LIN {X 0,Y 369.158,Z 304.498,A -85,B 0,C 180,E1 -12863.442,E2 -12863.442} C_VEL
LIN {X 0,Y 369.295,Z 304.483,A -85,B 0,C 180,E1 -12867.819,E2 -12867.819} C_VEL
LIN {X 0,Y 369.206,Z 304.491,A -85,B 0,C 180,E1 -12871.091,E2 -12871.091} C_VEL
LIN {X 0,Y 369.294,Z 304.487,A -85,B 0,C 180,E1 -12872.182,E2 -12872.182} C_VEL
LIN {X 0,Y 369.16,Z 304.501,A -85,B 0,C 180,E1 -12876.56,E2 -12876.56} C_VEL
LIN {X 0,Y 369.039,Z 304.513,A -85,B 0,C 180,E1 -12879.87,E2 -12879.87} C_VEL
LIN {X 0,Y 369.006,Z 304.516,A -85,B 0,C 180,E1 -12883.749,E2 -12883.749} C_VEL
LIN {X 0,Y 368.958,Z 304.522,A -85,B 0,C 180,E1 -12887.745,E2 -12887.745} C_VEL
LIN {X 0,Y 368.914,Z 304.532,A -85,B 0,C 180,E1 -12891.221,E2 -12891.221} C_VEL
LIN {X 0,Y 368.962,Z 304.615,A -85,B 0,C 180,E1 -12893.171,E2 -12893.171} C_VEL
LIN {X 0,Y 370.807,Z 314.362,A -85,B 0,C 180,E1 -12895.845,E2 -12895.845} C_VEL
LIN {X 0,Y 373.154,Z 322.489,A -85,B 0,C 180,E1 -12896.158,E2 -12896.158} C_VEL
LIN {X 0,Y 376.257,Z 338.846,A -85,B 0,C 180,E1 -12896.672,E2 -12896.672} C_VEL
LIN {X 0,Y 374.9,Z 409.964,A -85,B 0,C 180,E1 -12898.135,E2 -12898.135} C_VEL
LIN {X 0,Y 374.138,Z 415.804,A -85,B 0,C 180,E1 -12898.226,E2 -12898.226} C_VEL
LIN {X 0,Y 371.004,Z 425.22,A -85,B 0,C 180,E1 -12898.352,E2 -12898.352} C_VEL
LIN {X 0,Y 367.894,Z 434.497,A -85,B 0,C 180,E1 -12898.587,E2 -12898.587} C_VEL
LIN {X 0,Y 367.116,Z 440.104,A -85,B 0,C 180,E1 -12898.842,E2 -12898.842} C_VEL
LIN {X 0,Y 366.35,Z 452.424,A -85,B 0,C 180,E1 -12899.603,E2 -12899.603} C_VEL
LIN {X 0,Y 365.516,Z 464,A -85,B 0,C 180,E1 -12900.548,E2 -12900.548} C_VEL
LIN {X 0,Y 364.656,Z 474.566,A -85,B 0,C 180,E1 -12901.646,E2 -12901.646} C_VEL
LIN {X 0,Y 363.853,Z 484.377,A -85,B 0,C 180,E1 -12902.905,E2 -12902.905} C_VEL
LIN {X 0,Y 362.988,Z 493.439,A -85,B 0,C 180,E1 -12904.327,E2 -12904.327} C_VEL
LIN {X 0,Y 362.136,Z 501.792,A -85,B 0,C 180,E1 -12905.949,E2 -12905.949} C_VEL
LIN {X 0,Y 361.431,Z 509.337,A -85,B 0,C 180,E1 -12907.799,E2 -12907.799} C_VEL
LIN {X 0,Y 361.041,Z 514.472,A -85,B 0,C 180,E1 -12909.389,E2 -12909.389} C_VEL
LIN {X 0,Y 360.728,Z 518.553,A -85,B 0,C 180,E1 -12910.99,E2 -12910.99} C_VEL
LIN {X 0,Y 360.364,Z 522.397,A -85,B 0,C 180,E1 -12913.047,E2 -12913.047} C_VEL
LIN {X 0,Y 360.207,Z 524.3,A -85,B 0,C 180,E1 -12914.62,E2 -12914.62} C_VEL
LIN {X 0,Y 360.172,Z 525.614,A -85,B 0,C 180,E1 -12916.925,E2 -12916.925} C_VEL
LIN {X 0,Y 360.174,Z 525.57,A -85,B 0,C 180,E1 -12918.437,E2 -12918.437} C_VEL
LIN {X 0,Y 360.258,Z 524.77,A -85,B 0,C 180,E1 -12919.926,E2 -12919.926} C_VEL
LIN {X 0,Y 360.63,Z 522.252,A -85,B 0,C 180,E1 -12922.129,E2 -12922.129} C_VEL
LIN {X 0,Y 361.086,Z 518.191,A -85,B 0,C 180,E1 -12924.274,E2 -12924.274} C_VEL
LIN {X 0,Y 361.701,Z 513.027,A -85,B 0,C 180,E1 -12926.201,E2 -12926.201} C_VEL
LIN {X 0,Y 362.518,Z 506.261,A -85,B 0,C 180,E1 -12928.11,E2 -12928.11} C_VEL
LIN {X 0,Y 363.46,Z 498.606,A -85,B 0,C 180,E1 -12929.818,E2 -12929.818} C_VEL
LIN {X 0,Y 364.603,Z 489.19,A -85,B 0,C 180,E1 -12931.477,E2 -12931.477} C_VEL
LIN {X 0,Y 365.673,Z 479.6,A -85,B 0,C 180,E1 -12932.841,E2 -12932.841} C_VEL
LIN {X 0,Y 366.845,Z 468.816,A -85,B 0,C 180,E1 -12934.07,E2 -12934.07} C_VEL
LIN {X 0,Y 367.921,Z 456.729,A -85,B 0,C 180,E1 -12935.15,E2 -12935.15} C_VEL
LIN {X 0,Y 368.805,Z 445.404,A -85,B 0,C 180,E1 -12935.928,E2 -12935.928} C_VEL
LIN {X 0,Y 369.489,Z 432.429,A -85,B 0,C 180,E1 -12936.586,E2 -12936.586} C_VEL
LIN {X 0,Y 369.985,Z 418.805,A -85,B 0,C 180,E1 -12937.027,E2 -12937.027} C_VEL
LIN {X 0,Y 371.953,Z 339.841,A -85,B 0,C 180,E1 -12938.741,E2 -12938.741} C_VEL
LIN {X 0,Y 369.024,Z 326.317,A -85,B 0,C 180,E1 -12939.288,E2 -12939.288} C_VEL
LIN {X 0,Y 364.19,Z 314.682,A -85,B 0,C 180,E1 -12939.968,E2 -12939.968} C_VEL
LIN {X 0,Y 361.958,Z 305.404,A -85,B 0,C 180,E1 -12942.326,E2 -12942.326} C_VEL
LIN {X 0,Y 362.001,Z 305.397,A -85,B 0,C 180,E1 -12946.101,E2 -12946.101} C_VEL
LIN {X 0,Y 362.033,Z 305.389,A -85,B 0,C 180,E1 -12949.938,E2 -12949.938} C_VEL
LIN {X 0,Y 362.153,Z 305.376,A -85,B 0,C 180,E1 -12952.192,E2 -12952.192} C_VEL
LIN {X 0,Y 362.118,Z 305.379,A -85,B 0,C 180,E1 -12954.431,E2 -12954.431} C_VEL
LIN {X 0,Y 362.282,Z 305.358,A -85,B 0,C 180,E1 -12957.776,E2 -12957.776} C_VEL
LIN {X 0,Y 362.428,Z 305.34,A -85,B 0,C 180,E1 -12960,E2 -12960} C_VEL
LIN {X 0,Y 362.282,Z 305.36,A -85,B 0,C 180,E1 -12962.223,E2 -12962.223} C_VEL
LIN {X 0,Y 362.141,Z 305.368,A -85,B 0,C 180,E1 -12966.687,E2 -12966.687} C_VEL
LIN {X 0,Y 362.033,Z 305.384,A -85,B 0,C 180,E1 -12970.062,E2 -12970.062} C_VEL
LIN {X 0,Y 362,Z 305.386,A -85,B 0,C 180,E1 -12973.898,E2 -12973.898} C_VEL
LIN {X 0,Y 361.93,Z 305.394,A -85,B 0,C 180,E1 -12976.934,E2 -12976.934} C_VEL
LIN {X 0,Y 361.888,Z 305.402,A -85,B 0,C 180,E1 -12980.461,E2 -12980.461} C_VEL
LIN {X 0,Y 361.895,Z 305.401,A -85,B 0,C 180,E1 -12984.113,E2 -12984.113} C_VEL
LIN {X 0,Y 361.943,Z 305.399,A -85,B 0,C 180,E1 -12986.721,E2 -12986.721} C_VEL
LIN {X 0,Y 361.875,Z 305.407,A -85,B 0,C 180,E1 -12990.328,E2 -12990.328} C_VEL
LIN {X 0,Y 361.856,Z 305.408,A -85,B 0,C 180,E1 -12994.28,E2 -12994.28} C_VEL
LIN {X 0,Y 361.865,Z 305.407,A -85,B 0,C 180,E1 -12997.223,E2 -12997.223} C_VEL
LIN {X 0,Y 361.837,Z 305.41,A -85,B 0,C 180,E1 -13000.755,E2 -13000.755} C_VEL
LIN {X 0,Y 361.819,Z 305.415,A -85,B 0,C 180,E1 -13004.368,E2 -13004.368} C_VEL
LIN {X 0,Y 361.838,Z 305.413,A -85,B 0,C 180,E1 -13007.568,E2 -13007.568} C_VEL
LIN {X 0,Y 361.87,Z 305.41,A -85,B 0,C 180,E1 -13010.973,E2 -13010.973} C_VEL
LIN {X 0,Y 361.876,Z 305.413,A -85,B 0,C 180,E1 -13014.655,E2 -13014.655} C_VEL
LIN {X 0,Y 361.84,Z 305.417,A -85,B 0,C 180,E1 -13018.37,E2 -13018.37} C_VEL
LIN {X 0,Y 361.934,Z 305.557,A -85,B 0,C 180,E1 -13019.41,E2 -13019.41} C_VEL
LIN {X 0,Y 364.728,Z 317.304,A -85,B 0,C 180,E1 -13022.422,E2 -13022.422} C_VEL
LIN {X 0,Y 366.195,Z 325.557,A -85,B 0,C 180,E1 -13024.425,E2 -13024.425} C_VEL
LIN {X 0,Y 365.204,Z 338.309,A -85,B 0,C 180,E1 -13027.185,E2 -13027.185} C_VEL
LIN {X 0,Y 369.361,Z 360.306,A -85,B 0,C 180,E1 -13028.032,E2 -13028.032} C_VEL
LIN {X 0,Y 371.307,Z 374.136,A -85,B 0,C 180,E1 -13028.503,E2 -13028.503} C_VEL
LIN {X 0,Y 369.57,Z 448.21,A -85,B 0,C 180,E1 -13030.127,E2 -13030.127} C_VEL
LIN {X 0,Y 368.75,Z 462.309,A -85,B 0,C 180,E1 -13030.661,E2 -13030.661} C_VEL
LIN {X 0,Y 367.815,Z 474.39,A -85,B 0,C 180,E1 -13031.334,E2 -13031.334} C_VEL
LIN {X 0,Y 366.667,Z 486.939,A -85,B 0,C 180,E1 -13032.285,E2 -13032.285} C_VEL
LIN {X 0,Y 365.455,Z 498.198,A -85,B 0,C 180,E1 -13033.377,E2 -13033.377} C_VEL
LIN {X 0,Y 364.303,Z 508.998,A -85,B 0,C 180,E1 -13034.706,E2 -13034.706} C_VEL
LIN {X 0,Y 363.353,Z 517.608,A -85,B 0,C 180,E1 -13036.008,E2 -13036.008} C_VEL
LIN {X 0,Y 362.265,Z 526.631,A -85,B 0,C 180,E1 -13037.678,E2 -13037.678} C_VEL
LIN {X 0,Y 361.447,Z 533.915,A -85,B 0,C 180,E1 -13039.355,E2 -13039.355} C_VEL
LIN {X 0,Y 360.915,Z 539.734,A -85,B 0,C 180,E1 -13041.037,E2 -13041.037} C_VEL
LIN {X 0,Y 360.591,Z 544.332,A -85,B 0,C 180,E1 -13042.721,E2 -13042.721} C_VEL
LIN {X 0,Y 360.383,Z 547.831,A -85,B 0,C 180,E1 -13044.404,E2 -13044.404} C_VEL
LIN {X 0,Y 360.365,Z 549.58,A -85,B 0,C 180,E1 -13045.525,E2 -13045.525} C_VEL
LIN {X 0,Y 360.302,Z 550.917,A -85,B 0,C 180,E1 -13046.645,E2 -13046.645} C_VEL
LIN {X 0,Y 360.297,Z 551.851,A -85,B 0,C 180,E1 -13047.764,E2 -13047.764} C_VEL
LIN {X 0,Y 360.369,Z 552.338,A -85,B 0,C 180,E1 -13048.882,E2 -13048.882} C_VEL
LIN {X 0,Y 360.424,Z 552.415,A -85,B 0,C 180,E1 -13049.999,E2 -13049.999} C_VEL
LIN {X 0,Y 360.385,Z 552.091,A -85,B 0,C 180,E1 -13051.117,E2 -13051.117} C_VEL
LIN {X 0,Y 360.304,Z 551.362,A -85,B 0,C 180,E1 -13052.235,E2 -13052.235} C_VEL
LIN {X 0,Y 360.305,Z 550.176,A -85,B 0,C 180,E1 -13053.354,E2 -13053.354} C_VEL
LIN {X 0,Y 360.364,Z 547.607,A -85,B 0,C 180,E1 -13055.034,E2 -13055.034} C_VEL
LIN {X 0,Y 360.496,Z 543.988,A -85,B 0,C 180,E1 -13056.717,E2 -13056.717} C_VEL
LIN {X 0,Y 360.747,Z 539.221,A -85,B 0,C 180,E1 -13058.401,E2 -13058.401} C_VEL
LIN {X 0,Y 361.25,Z 532.028,A -85,B 0,C 180,E1 -13060.366,E2 -13060.366} C_VEL
LIN {X 0,Y 361.951,Z 524.189,A -85,B 0,C 180,E1 -13062.047,E2 -13062.047} C_VEL
LIN {X 0,Y 362.661,Z 516.147,A -85,B 0,C 180,E1 -13063.446,E2 -13063.446} C_VEL
LIN {X 0,Y 363.64,Z 505.802,A -85,B 0,C 180,E1 -13064.908,E2 -13064.908} C_VEL
LIN {X 0,Y 364.478,Z 495.426,A -85,B 0,C 180,E1 -13066.091,E2 -13066.091} C_VEL
LIN {X 0,Y 365.404,Z 484.808,A -85,B 0,C 180,E1 -13067.055,E2 -13067.055} C_VEL
LIN {X 0,Y 366.352,Z 472.083,A -85,B 0,C 180,E1 -13067.946,E2 -13067.946} C_VEL
LIN {X 0,Y 367.178,Z 459.469,A -85,B 0,C 180,E1 -13068.59,E2 -13068.59} C_VEL
LIN {X 0,Y 367.723,Z 446.201,A -85,B 0,C 180,E1 -13069.032,E2 -13069.032} C_VEL
LIN {X 0,Y 368.945,Z 372.876,A -85,B 0,C 180,E1 -13070.593,E2 -13070.593} C_VEL
LIN {X 0,Y 364.224,Z 340.195,A -85,B 0,C 180,E1 -13071.604,E2 -13071.604} C_VEL
LIN {X 0,Y 365.627,Z 325.106,A -85,B 0,C 180,E1 -13075.016,E2 -13075.016} C_VEL
LIN {X 0,Y 364.637,Z 318.571,A -85,B 0,C 180,E1 -13076.601,E2 -13076.601} C_VEL
LIN {X 0,Y 362.081,Z 306.333,A -85,B 0,C 180,E1 -13079.706,E2 -13079.706} C_VEL
LIN {X 0,Y 361.886,Z 305.409,A -85,B 0,C 180,E1 -13079.949,E2 -13079.949} C_VEL
LIN {X 0,Y 361.858,Z 305.409,A -85,B 0,C 180,E1 -13083.369,E2 -13083.369} C_VEL
LIN {X 0,Y 361.864,Z 305.406,A -85,B 0,C 180,E1 -13087.017,E2 -13087.017} C_VEL
LIN {X 0,Y 361.851,Z 305.409,A -85,B 0,C 180,E1 -13089.861,E2 -13089.861} C_VEL
LIN {X 0,Y 361.832,Z 305.412,A -85,B 0,C 180,E1 -13092.828,E2 -13092.828} C_VEL
LIN {X 0,Y 361.816,Z 305.413,A -85,B 0,C 180,E1 -13095.946,E2 -13095.946} C_VEL
LIN {X 0,Y 361.833,Z 305.41,A -85,B 0,C 180,E1 -13099.244,E2 -13099.244} C_VEL
LIN {X 0,Y 361.867,Z 305.411,A -85,B 0,C 180,E1 -13102.775,E2 -13102.775} C_VEL
LIN {X 0,Y 361.849,Z 305.407,A -85,B 0,C 180,E1 -13105.719,E2 -13105.719} C_VEL
LIN {X 0,Y 361.868,Z 305.405,A -85,B 0,C 180,E1 -13109.672,E2 -13109.672} C_VEL
LIN {X 0,Y 361.948,Z 305.397,A -85,B 0,C 180,E1 -13113.475,E2 -13113.475} C_VEL
LIN {X 0,Y 361.885,Z 305.41,A -85,B 0,C 180,E1 -13117.144,E2 -13117.144} C_VEL
LIN {X 0,Y 361.915,Z 305.401,A -85,B 0,C 180,E1 -13120.724,E2 -13120.724} C_VEL
LIN {X 0,Y 361.94,Z 305.396,A -85,B 0,C 180,E1 -13124.226,E2 -13124.226} C_VEL
LIN {X 0,Y 361.993,Z 305.39,A -85,B 0,C 180,E1 -13126.528,E2 -13126.528} C_VEL
LIN {X 0,Y 362.025,Z 305.387,A -85,B 0,C 180,E1 -13129.938,E2 -13129.938} C_VEL
LIN {X 0,Y 362.145,Z 305.371,A -85,B 0,C 180,E1 -13132.193,E2 -13132.193} C_VEL
LIN {X 0,Y 362.112,Z 305.375,A -85,B 0,C 180,E1 -13134.431,E2 -13134.431} C_VEL
LIN {X 0,Y 362.274,Z 305.36,A -85,B 0,C 180,E1 -13137.777,E2 -13137.777} C_VEL
LIN {X 0,Y 362.42,Z 305.34,A -85,B 0,C 180,E1 -13140,E2 -13140} C_VEL
LIN {X 0,Y 362.275,Z 305.357,A -85,B 0,C 180,E1 -13142.224,E2 -13142.224} C_VEL
LIN {X 0,Y 362.134,Z 305.372,A -85,B 0,C 180,E1 -13146.687,E2 -13146.687} C_VEL
LIN {X 0,Y 362.026,Z 305.392,A -85,B 0,C 180,E1 -13150.063,E2 -13150.063} C_VEL
LIN {X 0,Y 361.993,Z 305.394,A -85,B 0,C 180,E1 -13153.899,E2 -13153.899} C_VEL
LIN {X 0,Y 361.963,Z 305.397,A -85,B 0,C 180,E1 -13157.939,E2 -13157.939} C_VEL
LIN {X 0,Y 361.856,Z 305.407,A -85,B 0,C 180,E1 -13161.656,E2 -13161.656} C_VEL
LIN {X 0,Y 361.886,Z 305.403,A -85,B 0,C 180,E1 -13165.294,E2 -13165.294} C_VEL
LIN {X 0,Y 361.851,Z 305.409,A -85,B 0,C 180,E1 -13169.075,E2 -13169.075} C_VEL
LIN {X 0,Y 361.845,Z 305.411,A -85,B 0,C 180,E1 -13172.946,E2 -13172.946} C_VEL
LIN {X 0,Y 361.865,Z 305.405,A -85,B 0,C 180,E1 -13175.638,E2 -13175.638} C_VEL
LIN {X 0,Y 361.83,Z 305.414,A -85,B 0,C 180,E1 -13179.02,E2 -13179.02} C_VEL
LIN {X 0,Y 361.833,Z 305.416,A -85,B 0,C 180,E1 -13182.83,E2 -13182.83} C_VEL
LIN {X 0,Y 361.815,Z 305.412,A -85,B 0,C 180,E1 -13185.948,E2 -13185.948} C_VEL
LIN {X 0,Y 361.811,Z 305.417,A -85,B 0,C 180,E1 -13189.25,E2 -13189.25} C_VEL
LIN {X 0,Y 361.864,Z 305.41,A -85,B 0,C 180,E1 -13192.983,E2 -13192.983} C_VEL
LIN {X 0,Y 361.859,Z 305.407,A -85,B 0,C 180,E1 -13196.632,E2 -13196.632} C_VEL
LIN {X 0,Y 361.856,Z 305.41,A -85,B 0,C 180,E1 -13199.671,E2 -13199.671} C_VEL
LIN {X 0,Y 361.857,Z 305.413,A -85,B 0,C 180,E1 -13203.468,E2 -13203.468} C_VEL
LIN {X 0,Y 361.878,Z 305.406,A -85,B 0,C 180,E1 -13207.145,E2 -13207.145} C_VEL
LIN {X 0,Y 361.889,Z 305.402,A -85,B 0,C 180,E1 -13210.723,E2 -13210.723} C_VEL
LIN {X 0,Y 361.946,Z 305.397,A -85,B 0,C 180,E1 -13214.227,E2 -13214.227} C_VEL
LIN {X 0,Y 362.002,Z 305.389,A -85,B 0,C 180,E1 -13216.529,E2 -13216.529} C_VEL
LIN {X 0,Y 361.998,Z 305.396,A -85,B 0,C 180,E1 -13219.938,E2 -13219.938} C_VEL
LIN {X 0,Y 362.122,Z 305.374,A -85,B 0,C 180,E1 -13223.314,E2 -13223.314} C_VEL
LIN {X 0,Y 362.257,Z 305.36,A -85,B 0,C 180,E1 -13227.777,E2 -13227.777} C_VEL
LIN {X 0,Y 362.177,Z 305.367,A -85,B 0,C 180,E1 -13231.113,E2 -13231.113} C_VEL
LIN {X 0,Y 362.256,Z 305.364,A -85,B 0,C 180,E1 -13232.224,E2 -13232.224} C_VEL
LIN {X 0,Y 362.124,Z 305.376,A -85,B 0,C 180,E1 -13236.688,E2 -13236.688} C_VEL
LIN {X 0,Y 361.981,Z 305.394,A -85,B 0,C 180,E1 -13240.064,E2 -13240.064} C_VEL
LIN {X 0,Y 361.955,Z 305.395,A -85,B 0,C 180,E1 -13243.868,E2 -13243.868} C_VEL
LIN {X 0,Y 361.909,Z 305.4,A -85,B 0,C 180,E1 -13247.907,E2 -13247.907} C_VEL
LIN {X 0,Y 361.866,Z 305.41,A -85,B 0,C 180,E1 -13251.655,E2 -13251.655} C_VEL
LIN {X 0,Y 361.922,Z 305.534,A -85,B 0,C 180,E1 -13252.929,E2 -13252.929} C_VEL
LIN {X 0,Y 363.666,Z 314.598,A -85,B 0,C 180,E1 -13255.467,E2 -13255.467} C_VEL
LIN {X 0,Y 366.545,Z 324.082,A -85,B 0,C 180,E1 -13255.85,E2 -13255.85} C_VEL
LIN {X 0,Y 369.521,Z 340.035,A -85,B 0,C 180,E1 -13256.362,E2 -13256.362} C_VEL
LIN {X 0,Y 367.809,Z 422.701,A -85,B 0,C 180,E1 -13258.127,E2 -13258.127} C_VEL
LIN {X 0,Y 367.192,Z 436.734,A -85,B 0,C 180,E1 -13258.666,E2 -13258.666} C_VEL
LIN {X 0,Y 367.116,Z 440.104,A -85,B 0,C 180,E1 -13258.842,E2 -13258.842} C_VEL
LIN {X 0,Y 366.281,Z 445.703,A -85,B 0,C 180,E1 -13259.135,E2 -13259.135} C_VEL
LIN {X 0,Y 362.982,Z 454.586,A -85,B 0,C 180,E1 -13259.625,E2 -13259.625} C_VEL
LIN {X 0,Y 359.464,Z 463.074,A -85,B 0,C 180,E1 -13260.21,E2 -13260.21} C_VEL
LIN {X 0,Y 358.319,Z 468.05,A -85,B 0,C 180,E1 -13260.66,E2 -13260.66} C_VEL
LIN {X 0,Y 357.412,Z 478.87,A -85,B 0,C 180,E1 -13261.902,E2 -13261.902} C_VEL
LIN {X 0,Y 356.445,Z 488.979,A -85,B 0,C 180,E1 -13263.345,E2 -13263.345} C_VEL
LIN {X 0,Y 355.546,Z 498.18,A -85,B 0,C 180,E1 -13264.977,E2 -13264.977} C_VEL
LIN {X 0,Y 354.731,Z 506,A -85,B 0,C 180,E1 -13266.72,E2 -13266.72} C_VEL
LIN {X 0,Y 354.103,Z 512.699,A -85,B 0,C 180,E1 -13268.604,E2 -13268.604} C_VEL
LIN {X 0,Y 353.782,Z 517.133,A -85,B 0,C 180,E1 -13270.201,E2 -13270.201} C_VEL
LIN {X 0,Y 353.523,Z 520.513,A -85,B 0,C 180,E1 -13271.758,E2 -13271.758} C_VEL
LIN {X 0,Y 353.22,Z 523.095,A -85,B 0,C 180,E1 -13273.349,E2 -13273.349} C_VEL
LIN {X 0,Y 353.145,Z 524.166,A -85,B 0,C 180,E1 -13274.238,E2 -13274.238} C_VEL
LIN {X 0,Y 353.061,Z 525.47,A -85,B 0,C 180,E1 -13275.836,E2 -13275.836} C_VEL
LIN {X 0,Y 353.079,Z 525.963,A -85,B 0,C 180,E1 -13277.433,E2 -13277.433} C_VEL
LIN {X 0,Y 353.124,Z 525.594,A -85,B 0,C 180,E1 -13279.139,E2 -13279.139} C_VEL
LIN {X 0,Y 353.297,Z 524.285,A -85,B 0,C 180,E1 -13280.879,E2 -13280.879} C_VEL
LIN {X 0,Y 353.656,Z 521.964,A -85,B 0,C 180,E1 -13282.646,E2 -13282.646} C_VEL
LIN {X 0,Y 354.083,Z 518.475,A -85,B 0,C 180,E1 -13284.468,E2 -13284.468} C_VEL
LIN {X 0,Y 354.68,Z 513.647,A -85,B 0,C 180,E1 -13286.329,E2 -13286.329} C_VEL
LIN {X 0,Y 355.511,Z 507.201,A -85,B 0,C 180,E1 -13288.218,E2 -13288.218} C_VEL
LIN {X 0,Y 356.468,Z 499.745,A -85,B 0,C 180,E1 -13289.946,E2 -13289.946} C_VEL
LIN {X 0,Y 357.599,Z 491.207,A -85,B 0,C 180,E1 -13291.536,E2 -13291.536} C_VEL
LIN {X 0,Y 358.825,Z 480.892,A -85,B 0,C 180,E1 -13293.068,E2 -13293.068} C_VEL
LIN {X 0,Y 360.102,Z 469.871,A -85,B 0,C 180,E1 -13294.371,E2 -13294.371} C_VEL
LIN {X 0,Y 361.182,Z 458.584,A -85,B 0,C 180,E1 -13295.422,E2 -13295.422} C_VEL
LIN {X 0,Y 362.237,Z 445.777,A -85,B 0,C 180,E1 -13296.336,E2 -13296.336} C_VEL
LIN {X 0,Y 362.951,Z 432.861,A -85,B 0,C 180,E1 -13297.008,E2 -13297.008} C_VEL
LIN {X 0,Y 363.476,Z 418.992,A -85,B 0,C 180,E1 -13297.467,E2 -13297.467} C_VEL
LIN {X 0,Y 365.552,Z 340.931,A -85,B 0,C 180,E1 -13299.2,E2 -13299.2} C_VEL
LIN {X 0,Y 362.919,Z 328.903,A -85,B 0,C 180,E1 -13299.701,E2 -13299.701} C_VEL
LIN {X 0,Y 357.064,Z 314.924,A -85,B 0,C 180,E1 -13300.581,E2 -13300.581} C_VEL
LIN {X 0,Y 354.896,Z 306.284,A -85,B 0,C 180,E1 -13302.868,E2 -13302.868} C_VEL
LIN {X 0,Y 354.954,Z 306.274,A -85,B 0,C 180,E1 -13306.255,E2 -13306.255} C_VEL
LIN {X 0,Y 354.98,Z 306.267,A -85,B 0,C 180,E1 -13309.736,E2 -13309.736} C_VEL
LIN {X 0,Y 355.116,Z 306.251,A -85,B 0,C 180,E1 -13312.037,E2 -13312.037} C_VEL
LIN {X 0,Y 355.093,Z 306.255,A -85,B 0,C 180,E1 -13314.32,E2 -13314.32} C_VEL
LIN {X 0,Y 355.245,Z 306.234,A -85,B 0,C 180,E1 -13317.732,E2 -13317.732} C_VEL
LIN {X 0,Y 355.377,Z 306.218,A -85,B 0,C 180,E1 -13320,E2 -13320} C_VEL
LIN {X 0,Y 355.245,Z 306.236,A -85,B 0,C 180,E1 -13322.267,E2 -13322.267} C_VEL
LIN {X 0,Y 355.105,Z 306.244,A -85,B 0,C 180,E1 -13326.82,E2 -13326.82} C_VEL
LIN {X 0,Y 354.979,Z 306.262,A -85,B 0,C 180,E1 -13330.264,E2 -13330.264} C_VEL
LIN {X 0,Y 354.945,Z 306.265,A -85,B 0,C 180,E1 -13334.018,E2 -13334.018} C_VEL
LIN {X 0,Y 354.891,Z 306.272,A -85,B 0,C 180,E1 -13338.092,E2 -13338.092} C_VEL
LIN {X 0,Y 354.819,Z 306.283,A -85,B 0,C 180,E1 -13342.107,E2 -13342.107} C_VEL
LIN {X 0,Y 354.9,Z 306.273,A -85,B 0,C 180,E1 -13345.827,E2 -13345.827} C_VEL
LIN {X 0,Y 354.819,Z 306.285,A -85,B 0,C 180,E1 -13349.682,E2 -13349.682} C_VEL
LIN {X 0,Y 354.808,Z 306.286,A -85,B 0,C 180,E1 -13353.702,E2 -13353.702} C_VEL
LIN {X 0,Y 354.799,Z 306.289,A -85,B 0,C 180,E1 -13356.459,E2 -13356.459} C_VEL
LIN {X 0,Y 354.826,Z 306.288,A -85,B 0,C 180,E1 -13359.423,E2 -13359.423} C_VEL
LIN {X 0,Y 354.79,Z 306.292,A -85,B 0,C 180,E1 -13362.867,E2 -13362.867} C_VEL
LIN {X 0,Y 354.769,Z 306.292,A -85,B 0,C 180,E1 -13366.103,E2 -13366.103} C_VEL
LIN {X 0,Y 354.79,Z 306.292,A -85,B 0,C 180,E1 -13369.179,E2 -13369.179} C_VEL
LIN {X 0,Y 354.809,Z 306.292,A -85,B 0,C 180,E1 -13372.402,E2 -13372.402} C_VEL
LIN {X 0,Y 354.814,Z 306.293,A -85,B 0,C 180,E1 -13374.941,E2 -13374.941} C_VEL
LIN {X 0,Y 354.842,Z 306.444,A -85,B 0,C 180,E1 -13378.896,E2 -13378.896} C_VEL
LIN {X 0,Y 357.597,Z 317.562,A -85,B 0,C 180,E1 -13381.856,E2 -13381.856} C_VEL
LIN {X 0,Y 359.322,Z 326.642,A -85,B 0,C 180,E1 -13384.121,E2 -13384.121} C_VEL
LIN {X 0,Y 358.985,Z 332.405,A -85,B 0,C 180,E1 -13385.416,E2 -13385.416} C_VEL
LIN {X 0,Y 358.481,Z 337.891,A -85,B 0,C 180,E1 -13386.625,E2 -13386.625} C_VEL
LIN {X 0,Y 362.686,Z 359.618,A -85,B 0,C 180,E1 -13387.512,E2 -13387.512} C_VEL
LIN {X 0,Y 364.895,Z 375.884,A -85,B 0,C 180,E1 -13388.076,E2 -13388.076} C_VEL
LIN {X 0,Y 363.007,Z 448.56,A -85,B 0,C 180,E1 -13389.715,E2 -13389.715} C_VEL
LIN {X 0,Y 362.223,Z 461.704,A -85,B 0,C 180,E1 -13390.224,E2 -13390.224} C_VEL
LIN {X 0,Y 361.242,Z 473.877,A -85,B 0,C 180,E1 -13390.907,E2 -13390.907} C_VEL
LIN {X 0,Y 360.124,Z 485.692,A -85,B 0,C 180,E1 -13391.805,E2 -13391.805} C_VEL
LIN {X 0,Y 358.832,Z 497.127,A -85,B 0,C 180,E1 -13392.915,E2 -13392.915} C_VEL
LIN {X 0,Y 357.743,Z 506.416,A -85,B 0,C 180,E1 -13394.035,E2 -13394.035} C_VEL
LIN {X 0,Y 356.61,Z 515.997,A -85,B 0,C 180,E1 -13395.447,E2 -13395.447} C_VEL
LIN {X 0,Y 355.502,Z 525.245,A -85,B 0,C 180,E1 -13397.149,E2 -13397.149} C_VEL
LIN {X 0,Y 354.523,Z 532.72,A -85,B 0,C 180,E1 -13398.855,E2 -13398.855} C_VEL
LIN {X 0,Y 353.87,Z 539.602,A -85,B 0,C 180,E1 -13400.857,E2 -13400.857} C_VEL
LIN {X 0,Y 353.513,Z 544.165,A -85,B 0,C 180,E1 -13402.575,E2 -13402.575} C_VEL
LIN {X 0,Y 353.289,Z 547.636,A -85,B 0,C 180,E1 -13404.291,E2 -13404.291} C_VEL
LIN {X 0,Y 353.278,Z 549.374,A -85,B 0,C 180,E1 -13405.435,E2 -13405.435} C_VEL
LIN {X 0,Y 353.224,Z 550.7,A -85,B 0,C 180,E1 -13406.577,E2 -13406.577} C_VEL
LIN {X 0,Y 353.203,Z 551.612,A -85,B 0,C 180,E1 -13407.719,E2 -13407.719} C_VEL
LIN {X 0,Y 353.27,Z 552.076,A -85,B 0,C 180,E1 -13408.859,E2 -13408.859} C_VEL
LIN {X 0,Y 353.329,Z 552.14,A -85,B 0,C 180,E1 -13409.999,E2 -13409.999} C_VEL
LIN {X 0,Y 353.286,Z 551.801,A -85,B 0,C 180,E1 -13411.139,E2 -13411.139} C_VEL
LIN {X 0,Y 353.208,Z 551.046,A -85,B 0,C 180,E1 -13412.28,E2 -13412.28} C_VEL
LIN {X 0,Y 353.227,Z 549.836,A -85,B 0,C 180,E1 -13413.421,E2 -13413.421} C_VEL
LIN {X 0,Y 353.268,Z 547.231,A -85,B 0,C 180,E1 -13415.136,E2 -13415.136} C_VEL
LIN {X 0,Y 353.414,Z 543.572,A -85,B 0,C 180,E1 -13416.852,E2 -13416.852} C_VEL
LIN {X 0,Y 353.686,Z 538.762,A -85,B 0,C 180,E1 -13418.57,E2 -13418.57} C_VEL
LIN {X 0,Y 354.132,Z 532.656,A -85,B 0,C 180,E1 -13420.288,E2 -13420.288} C_VEL
LIN {X 0,Y 354.822,Z 525.04,A -85,B 0,C 180,E1 -13422.003,E2 -13422.003} C_VEL
LIN {X 0,Y 355.54,Z 517.252,A -85,B 0,C 180,E1 -13423.43,E2 -13423.43} C_VEL
LIN {X 0,Y 356.49,Z 507.755,A -85,B 0,C 180,E1 -13424.849,E2 -13424.849} C_VEL
LIN {X 0,Y 357.358,Z 497.186,A -85,B 0,C 180,E1 -13426.128,E2 -13426.128} C_VEL
LIN {X 0,Y 358.44,Z 485.483,A -85,B 0,C 180,E1 -13427.25,E2 -13427.25} C_VEL
LIN {X 0,Y 359.392,Z 473.051,A -85,B 0,C 180,E1 -13428.159,E2 -13428.159} C_VEL
LIN {X 0,Y 360.274,Z 460.107,A -85,B 0,C 180,E1 -13428.849,E2 -13428.849} C_VEL
LIN {X 0,Y 360.882,Z 447.66,A -85,B 0,C 180,E1 -13429.296,E2 -13429.296} C_VEL
LIN {X 0,Y 362.205,Z 373.941,A -85,B 0,C 180,E1 -13430.904,E2 -13430.904} C_VEL
LIN {X 0,Y 357.295,Z 340.118,A -85,B 0,C 180,E1 -13431.945,E2 -13431.945} C_VEL
LIN {X 0,Y 358.646,Z 325.877,A -85,B 0,C 180,E1 -13435.226,E2 -13435.226} C_VEL
LIN {X 0,Y 357.276,Z 317.775,A -85,B 0,C 180,E1 -13437.254,E2 -13437.254} C_VEL
LIN {X 0,Y 354.848,Z 306.285,A -85,B 0,C 180,E1 -13440.251,E2 -13440.251} C_VEL
LIN {X 0,Y 354.804,Z 306.288,A -85,B 0,C 180,E1 -13443.701,E2 -13443.701} C_VEL
LIN {X 0,Y 354.795,Z 306.291,A -85,B 0,C 180,E1 -13446.459,E2 -13446.459} C_VEL
LIN {X 0,Y 354.821,Z 306.283,A -85,B 0,C 180,E1 -13449.423,E2 -13449.423} C_VEL
LIN {X 0,Y 354.784,Z 306.29,A -85,B 0,C 180,E1 -13452.866,E2 -13452.866} C_VEL
LIN {X 0,Y 354.764,Z 306.292,A -85,B 0,C 180,E1 -13456.103,E2 -13456.103} C_VEL
LIN {X 0,Y 354.785,Z 306.289,A -85,B 0,C 180,E1 -13459.179,E2 -13459.179} C_VEL
LIN {X 0,Y 354.808,Z 306.288,A -85,B 0,C 180,E1 -13462.401,E2 -13462.401} C_VEL
LIN {X 0,Y 354.807,Z 306.289,A -85,B 0,C 180,E1 -13464.94,E2 -13464.94} C_VEL
LIN {X 0,Y 354.788,Z 306.289,A -85,B 0,C 180,E1 -13468.405,E2 -13468.405} C_VEL
LIN {X 0,Y 354.841,Z 306.281,A -85,B 0,C 180,E1 -13471.618,E2 -13471.618} C_VEL
LIN {X 0,Y 354.894,Z 306.274,A -85,B 0,C 180,E1 -13474.172,E2 -13474.172} C_VEL
LIN {X 0,Y 354.829,Z 306.282,A -85,B 0,C 180,E1 -13477.894,E2 -13477.894} C_VEL
LIN {X 0,Y 354.917,Z 306.272,A -85,B 0,C 180,E1 -13481.891,E2 -13481.891} C_VEL
LIN {X 0,Y 354.937,Z 306.269,A -85,B 0,C 180,E1 -13485.981,E2 -13485.981} C_VEL
LIN {X 0,Y 354.972,Z 306.268,A -85,B 0,C 180,E1 -13489.736,E2 -13489.736} C_VEL
LIN {X 0,Y 355.108,Z 306.249,A -85,B 0,C 180,E1 -13492.037,E2 -13492.037} C_VEL
LIN {X 0,Y 355.086,Z 306.25,A -85,B 0,C 180,E1 -13494.321,E2 -13494.321} C_VEL
LIN {X 0,Y 355.238,Z 306.237,A -85,B 0,C 180,E1 -13497.733,E2 -13497.733} C_VEL
LIN {X 0,Y 355.39,Z 306.216,A -85,B 0,C 180,E1 -13500,E2 -13500} C_VEL
LIN {X 0,Y 355.238,Z 306.233,A -85,B 0,C 180,E1 -13502.268,E2 -13502.268} C_VEL
LIN {X 0,Y 355.097,Z 306.248,A -85,B 0,C 180,E1 -13506.82,E2 -13506.82} C_VEL
LIN {X 0,Y 354.972,Z 306.268,A -85,B 0,C 180,E1 -13510.265,E2 -13510.265} C_VEL
LIN {X 0,Y 354.938,Z 306.274,A -85,B 0,C 180,E1 -13514.02,E2 -13514.02} C_VEL
LIN {X 0,Y 354.918,Z 306.276,A -85,B 0,C 180,E1 -13518.109,E2 -13518.109} C_VEL
LIN {X 0,Y 354.81,Z 306.289,A -85,B 0,C 180,E1 -13522.108,E2 -13522.108} C_VEL
LIN {X 0,Y 354.818,Z 306.284,A -85,B 0,C 180,E1 -13525.834,E2 -13525.834} C_VEL
LIN {X 0,Y 354.795,Z 306.286,A -85,B 0,C 180,E1 -13529.684,E2 -13529.684} C_VEL
LIN {X 0,Y 354.783,Z 306.291,A -85,B 0,C 180,E1 -13532.334,E2 -13532.334} C_VEL
LIN {X 0,Y 354.819,Z 306.283,A -85,B 0,C 180,E1 -13535.7,E2 -13535.7} C_VEL
LIN {X 0,Y 354.796,Z 306.287,A -85,B 0,C 180,E1 -13539.42,E2 -13539.42} C_VEL
LIN {X 0,Y 354.785,Z 306.294,A -85,B 0,C 180,E1 -13542.868,E2 -13542.868} C_VEL
LIN {X 0,Y 354.764,Z 306.29,A -85,B 0,C 180,E1 -13546.104,E2 -13546.104} C_VEL
LIN {X 0,Y 354.765,Z 306.295,A -85,B 0,C 180,E1 -13549.177,E2 -13549.177} C_VEL
LIN {X 0,Y 354.8,Z 306.286,A -85,B 0,C 180,E1 -13552.405,E2 -13552.405} C_VEL
LIN {X 0,Y 354.812,Z 306.288,A -85,B 0,C 180,E1 -13554.942,E2 -13554.942} C_VEL
LIN {X 0,Y 354.793,Z 306.286,A -85,B 0,C 180,E1 -13558.406,E2 -13558.406} C_VEL
LIN {X 0,Y 354.797,Z 306.29,A -85,B 0,C 180,E1 -13561.615,E2 -13561.615} C_VEL
LIN {X 0,Y 354.841,Z 306.286,A -85,B 0,C 180,E1 -13565.423,E2 -13565.423} C_VEL
LIN {X 0,Y 354.829,Z 306.284,A -85,B 0,C 180,E1 -13569.114,E2 -13569.114} C_VEL
LIN {X 0,Y 354.883,Z 306.275,A -85,B 0,C 180,E1 -13572.72,E2 -13572.72} C_VEL
LIN {X 0,Y 354.954,Z 306.268,A -85,B 0,C 180,E1 -13576.256,E2 -13576.256} C_VEL
LIN {X 0,Y 354.954,Z 306.271,A -85,B 0,C 180,E1 -13579.736,E2 -13579.736} C_VEL
LIN {X 0,Y 355.088,Z 306.25,A -85,B 0,C 180,E1 -13583.181,E2 -13583.181} C_VEL
LIN {X 0,Y 355.219,Z 306.236,A -85,B 0,C 180,E1 -13587.733,E2 -13587.733} C_VEL
LIN {X 0,Y 355.148,Z 306.242,A -85,B 0,C 180,E1 -13591.135,E2 -13591.135} C_VEL
LIN {X 0,Y 355.218,Z 306.24,A -85,B 0,C 180,E1 -13592.268,E2 -13592.268} C_VEL
LIN {X 0,Y 355.091,Z 306.251,A -85,B 0,C 180,E1 -13596.821,E2 -13596.821} C_VEL
LIN {X 0,Y 354.941,Z 306.273,A -85,B 0,C 180,E1 -13600.266,E2 -13600.266} C_VEL
LIN {X 0,Y 354.897,Z 306.275,A -85,B 0,C 180,E1 -13603.986,E2 -13603.986} C_VEL
LIN {X 0,Y 354.847,Z 306.281,A -85,B 0,C 180,E1 -13608.069,E2 -13608.069} C_VEL
LIN {X 0,Y 354.826,Z 306.288,A -85,B 0,C 180,E1 -13612.107,E2 -13612.107} C_VEL
LIN {X 0,Y 354.856,Z 306.342,A -85,B 0,C 180,E1 -13612.642,E2 -13612.642} C_VEL
LIN {X 0,Y 356.512,Z 314.884,A -85,B 0,C 180,E1 -13615.082,E2 -13615.082} C_VEL
LIN {X 0,Y 360.033,Z 326.234,A -85,B 0,C 180,E1 -13615.549,E2 -13615.549} C_VEL
LIN {X 0,Y 362.787,Z 340.967,A -85,B 0,C 180,E1 -13616.034,E2 -13616.034} C_VEL
LIN {X 0,Y 361.02,Z 422.602,A -85,B 0,C 180,E1 -13617.81,E2 -13617.81} C_VEL
LIN {X 0,Y 360.377,Z 436.598,A -85,B 0,C 180,E1 -13618.352,E2 -13618.352} C_VEL
LIN {X 0,Y 359.812,Z 448.771,A -85,B 0,C 180,E1 -13619.053,E2 -13619.053} C_VEL
LIN {X 0,Y 358.95,Z 460.503,A -85,B 0,C 180,E1 -13619.952,E2 -13619.952} C_VEL
LIN {X 0,Y 358.319,Z 468.05,A -85,B 0,C 180,E1 -13620.66,E2 -13620.66} C_VEL
LIN {X 0,Y 357.226,Z 472.998,A -85,B 0,C 180,E1 -13621.15,E2 -13621.15} C_VEL
LIN {X 0,Y 353.802,Z 480.724,A -85,B 0,C 180,E1 -13621.987,E2 -13621.987} C_VEL
LIN {X 0,Y 350.356,Z 487.935,A -85,B 0,C 180,E1 -13622.943,E2 -13622.943} C_VEL
LIN {X 0,Y 349.24,Z 492.074,A -85,B 0,C 180,E1 -13623.61,E2 -13623.61} C_VEL
LIN {X 0,Y 348.351,Z 499.888,A -85,B 0,C 180,E1 -13625.099,E2 -13625.099} C_VEL
LIN {X 0,Y 347.656,Z 506.706,A -85,B 0,C 180,E1 -13626.686,E2 -13626.686} C_VEL
LIN {X 0,Y 347.093,Z 512.49,A -85,B 0,C 180,E1 -13628.345,E2 -13628.345} C_VEL
LIN {X 0,Y 346.658,Z 518.175,A -85,B 0,C 180,E1 -13630.448,E2 -13630.448} C_VEL
LIN {X 0,Y 346.382,Z 521.386,A -85,B 0,C 180,E1 -13632.034,E2 -13632.034} C_VEL
LIN {X 0,Y 346.098,Z 523.788,A -85,B 0,C 180,E1 -13633.664,E2 -13633.664} C_VEL
LIN {X 0,Y 345.992,Z 525.371,A -85,B 0,C 180,E1 -13635.312,E2 -13635.312} C_VEL
LIN {X 0,Y 345.981,Z 526.146,A -85,B 0,C 180,E1 -13636.994,E2 -13636.994} C_VEL
LIN {X 0,Y 346.008,Z 526.068,A -85,B 0,C 180,E1 -13638.724,E2 -13638.724} C_VEL
LIN {X 0,Y 346.226,Z 524.577,A -85,B 0,C 180,E1 -13641.003,E2 -13641.003} C_VEL
LIN {X 0,Y 346.544,Z 522.694,A -85,B 0,C 180,E1 -13642.525,E2 -13642.525} C_VEL
LIN {X 0,Y 346.915,Z 519.919,A -85,B 0,C 180,E1 -13644.13,E2 -13644.13} C_VEL
LIN {X 0,Y 347.506,Z 515.483,A -85,B 0,C 180,E1 -13646.016,E2 -13646.016} C_VEL
LIN {X 0,Y 348.336,Z 509.565,A -85,B 0,C 180,E1 -13647.929,E2 -13647.929} C_VEL
LIN {X 0,Y 349.319,Z 502.173,A -85,B 0,C 180,E1 -13649.802,E2 -13649.802} C_VEL
LIN {X 0,Y 350.475,Z 494.186,A -85,B 0,C 180,E1 -13651.402,E2 -13651.402} C_VEL
LIN {X 0,Y 351.675,Z 484.742,A -85,B 0,C 180,E1 -13652.942,E2 -13652.942} C_VEL
LIN {X 0,Y 352.983,Z 474.074,A -85,B 0,C 180,E1 -13654.338,E2 -13654.338} C_VEL
LIN {X 0,Y 354.195,Z 462.825,A -85,B 0,C 180,E1 -13655.498,E2 -13655.498} C_VEL
LIN {X 0,Y 355.316,Z 451.388,A -85,B 0,C 180,E1 -13656.42,E2 -13656.42} C_VEL
LIN {X 0,Y 356.177,Z 438.53,A -85,B 0,C 180,E1 -13657.205,E2 -13657.205} C_VEL
LIN {X 0,Y 356.759,Z 426.989,A -85,B 0,C 180,E1 -13657.697,E2 -13657.697} C_VEL
LIN {X 0,Y 357.366,Z 408.297,A -85,B 0,C 180,E1 -13658.174,E2 -13658.174} C_VEL
LIN {X 0,Y 359.137,Z 341.8,A -85,B 0,C 180,E1 -13659.683,E2 -13659.683} C_VEL
LIN {X 0,Y 357.009,Z 331.885,A -85,B 0,C 180,E1 -13660.114,E2 -13660.114} C_VEL
LIN {X 0,Y 350.896,Z 317.694,A -85,B 0,C 180,E1 -13661.017,E2 -13661.017} C_VEL
LIN {X 0,Y 349.916,Z 315.313,A -85,B 0,C 180,E1 -13661.194,E2 -13661.194} C_VEL
LIN {X 0,Y 347.838,Z 307.164,A -85,B 0,C 180,E1 -13663.417,E2 -13663.417} C_VEL
LIN {X 0,Y 347.892,Z 307.153,A -85,B 0,C 180,E1 -13667.16,E2 -13667.16} C_VEL
LIN {X 0,Y 348.097,Z 307.124,A -85,B 0,C 180,E1 -13671.612,E2 -13671.612} C_VEL
LIN {X 0,Y 348.068,Z 307.13,A -85,B 0,C 180,E1 -13674.205,E2 -13674.205} C_VEL
LIN {X 0,Y 348.208,Z 307.111,A -85,B 0,C 180,E1 -13677.686,E2 -13677.686} C_VEL
LIN {X 0,Y 348.327,Z 307.096,A -85,B 0,C 180,E1 -13680,E2 -13680} C_VEL
LIN {X 0,Y 348.208,Z 307.112,A -85,B 0,C 180,E1 -13682.313,E2 -13682.313} C_VEL
LIN {X 0,Y 348.072,Z 307.12,A -85,B 0,C 180,E1 -13686.958,E2 -13686.958} C_VEL
LIN {X 0,Y 347.93,Z 307.14,A -85,B 0,C 180,E1 -13690.474,E2 -13690.474} C_VEL
LIN {X 0,Y 347.901,Z 307.143,A -85,B 0,C 180,E1 -13694.15,E2 -13694.15} C_VEL
LIN {X 0,Y 347.83,Z 307.153,A -85,B 0,C 180,E1 -13698.259,E2 -13698.259} C_VEL
LIN {X 0,Y 347.77,Z 307.16,A -85,B 0,C 180,E1 -13701.626,E2 -13701.626} C_VEL
LIN {X 0,Y 347.813,Z 307.155,A -85,B 0,C 180,E1 -13705.108,E2 -13705.108} C_VEL
LIN {X 0,Y 347.81,Z 307.151,A -85,B 0,C 180,E1 -13707.694,E2 -13707.694} C_VEL
LIN {X 0,Y 347.751,Z 307.167,A -85,B 0,C 180,E1 -13710.348,E2 -13710.348} C_VEL
LIN {X 0,Y 347.75,Z 307.164,A -85,B 0,C 180,E1 -13714.044,E2 -13714.044} C_VEL
LIN {X 0,Y 347.763,Z 307.163,A -85,B 0,C 180,E1 -13717.321,E2 -13717.321} C_VEL
LIN {X 0,Y 347.734,Z 307.167,A -85,B 0,C 180,E1 -13720.297,E2 -13720.297} C_VEL
LIN {X 0,Y 347.725,Z 307.17,A -85,B 0,C 180,E1 -13723.408,E2 -13723.408} C_VEL
LIN {X 0,Y 347.727,Z 307.17,A -85,B 0,C 180,E1 -13726.686,E2 -13726.686} C_VEL
LIN {X 0,Y 347.749,Z 307.167,A -85,B 0,C 180,E1 -13730.173,E2 -13730.173} C_VEL
LIN {X 0,Y 347.763,Z 307.17,A -85,B 0,C 180,E1 -13732.679,E2 -13732.679} C_VEL
LIN {X 0,Y 347.75,Z 307.175,A -85,B 0,C 180,E1 -13735.956,E2 -13735.956} C_VEL
LIN {X 0,Y 347.784,Z 307.273,A -85,B 0,C 180,E1 -13738.346,E2 -13738.346} C_VEL
LIN {X 0,Y 350.67,Z 318.82,A -85,B 0,C 180,E1 -13741.51,E2 -13741.51} C_VEL
LIN {X 0,Y 352.508,Z 328.46,A -85,B 0,C 180,E1 -13743.984,E2 -13743.984} C_VEL
LIN {X 0,Y 351.908,Z 336.315,A -85,B 0,C 180,E1 -13745.769,E2 -13745.769} C_VEL
LIN {X 0,Y 351.773,Z 337.663,A -85,B 0,C 180,E1 -13746.058,E2 -13746.058} C_VEL
LIN {X 0,Y 356.122,Z 359.52,A -85,B 0,C 180,E1 -13746.99,E2 -13746.99} C_VEL
LIN {X 0,Y 358.483,Z 376.745,A -85,B 0,C 180,E1 -13747.61,E2 -13747.61} C_VEL
LIN {X 0,Y 356.516,Z 448.261,A -85,B 0,C 180,E1 -13749.254,E2 -13749.254} C_VEL
LIN {X 0,Y 355.637,Z 462.083,A -85,B 0,C 180,E1 -13749.805,E2 -13749.805} C_VEL
LIN {X 0,Y 354.689,Z 473.492,A -85,B 0,C 180,E1 -13750.465,E2 -13750.465} C_VEL
LIN {X 0,Y 353.542,Z 484.514,A -85,B 0,C 180,E1 -13751.304,E2 -13751.304} C_VEL
LIN {X 0,Y 352.202,Z 496.075,A -85,B 0,C 180,E1 -13752.433,E2 -13752.433} C_VEL
LIN {X 0,Y 350.926,Z 506.561,A -85,B 0,C 180,E1 -13753.717,E2 -13753.717} C_VEL
LIN {X 0,Y 349.711,Z 516.054,A -85,B 0,C 180,E1 -13755.153,E2 -13755.153} C_VEL
LIN {X 0,Y 348.565,Z 525.245,A -85,B 0,C 180,E1 -13756.889,E2 -13756.889} C_VEL
LIN {X 0,Y 347.511,Z 532.678,A -85,B 0,C 180,E1 -13758.627,E2 -13758.627} C_VEL
LIN {X 0,Y 346.989,Z 537.723,A -85,B 0,C 180,E1 -13760.086,E2 -13760.086} C_VEL
LIN {X 0,Y 346.551,Z 542.639,A -85,B 0,C 180,E1 -13761.838,E2 -13761.838} C_VEL
LIN {X 0,Y 346.342,Z 545.305,A -85,B 0,C 180,E1 -13763.006,E2 -13763.006} C_VEL
LIN {X 0,Y 346.201,Z 547.455,A -85,B 0,C 180,E1 -13764.174,E2 -13764.174} C_VEL
LIN {X 0,Y 346.174,Z 549.175,A -85,B 0,C 180,E1 -13765.341,E2 -13765.341} C_VEL
LIN {X 0,Y 346.148,Z 550.484,A -85,B 0,C 180,E1 -13766.507,E2 -13766.507} C_VEL
LIN {X 0,Y 346.112,Z 551.369,A -85,B 0,C 180,E1 -13767.672,E2 -13767.672} C_VEL
LIN {X 0,Y 346.171,Z 551.816,A -85,B 0,C 180,E1 -13768.836,E2 -13768.836} C_VEL
LIN {X 0,Y 346.234,Z 551.865,A -85,B 0,C 180,E1 -13769.999,E2 -13769.999} C_VEL
LIN {X 0,Y 346.187,Z 551.51,A -85,B 0,C 180,E1 -13771.163,E2 -13771.163} C_VEL
LIN {X 0,Y 346.117,Z 550.725,A -85,B 0,C 180,E1 -13772.327,E2 -13772.327} C_VEL
LIN {X 0,Y 346.15,Z 549.497,A -85,B 0,C 180,E1 -13773.491,E2 -13773.491} C_VEL
LIN {X 0,Y 346.174,Z 546.439,A -85,B 0,C 180,E1 -13775.464,E2 -13775.464} C_VEL
LIN {X 0,Y 346.434,Z 541.697,A -85,B 0,C 180,E1 -13777.577,E2 -13777.577} C_VEL
LIN {X 0,Y 346.828,Z 535.397,A -85,B 0,C 180,E1 -13779.623,E2 -13779.623} C_VEL
LIN {X 0,Y 347.394,Z 528.513,A -85,B 0,C 180,E1 -13781.375,E2 -13781.375} C_VEL
LIN {X 0,Y 348.323,Z 519.937,A -85,B 0,C 180,E1 -13783.119,E2 -13783.119} C_VEL
LIN {X 0,Y 349.184,Z 511.186,A -85,B 0,C 180,E1 -13784.555,E2 -13784.555} C_VEL
LIN {X 0,Y 350.14,Z 500.411,A -85,B 0,C 180,E1 -13785.99,E2 -13785.99} C_VEL
LIN {X 0,Y 351.188,Z 489.27,A -85,B 0,C 180,E1 -13787.167,E2 -13787.167} C_VEL
LIN {X 0,Y 352.257,Z 477.083,A -85,B 0,C 180,E1 -13788.163,E2 -13788.163} C_VEL
LIN {X 0,Y 353.162,Z 464.419,A -85,B 0,C 180,E1 -13788.942,E2 -13788.942} C_VEL
LIN {X 0,Y 353.89,Z 450.955,A -85,B 0,C 180,E1 -13789.504,E2 -13789.504} C_VEL
LIN {X 0,Y 354.355,Z 431.18,A -85,B 0,C 180,E1 -13789.989,E2 -13789.989} C_VEL
LIN {X 0,Y 355.503,Z 375.103,A -85,B 0,C 180,E1 -13791.224,E2 -13791.224} C_VEL
LIN {X 0,Y 350.411,Z 339.838,A -85,B 0,C 180,E1 -13792.338,E2 -13792.338} C_VEL
LIN {X 0,Y 351.678,Z 326.861,A -85,B 0,C 180,E1 -13795.395,E2 -13795.395} C_VEL
LIN {X 0,Y 349.912,Z 317.071,A -85,B 0,C 180,E1 -13797.903,E2 -13797.903} C_VEL
LIN {X 0,Y 347.797,Z 307.16,A -85,B 0,C 180,E1 -13800.594,E2 -13800.594} C_VEL
LIN {X 0,Y 347.742,Z 307.169,A -85,B 0,C 180,E1 -13804.463,E2 -13804.463} C_VEL
LIN {X 0,Y 347.77,Z 307.165,A -85,B 0,C 180,E1 -13807.988,E2 -13807.988} C_VEL
LIN {X 0,Y 347.747,Z 307.165,A -85,B 0,C 180,E1 -13811.83,E2 -13811.83} C_VEL
LIN {X 0,Y 347.703,Z 307.171,A -85,B 0,C 180,E1 -13815.026,E2 -13815.026} C_VEL
LIN {X 0,Y 347.747,Z 307.169,A -85,B 0,C 180,E1 -13818.396,E2 -13818.396} C_VEL
LIN {X 0,Y 347.773,Z 307.162,A -85,B 0,C 180,E1 -13822.01,E2 -13822.01} C_VEL
LIN {X 0,Y 347.74,Z 307.165,A -85,B 0,C 180,E1 -13825.536,E2 -13825.536} C_VEL
LIN {X 0,Y 347.74,Z 307.166,A -85,B 0,C 180,E1 -13828.3,E2 -13828.3} C_VEL
LIN {X 0,Y 347.774,Z 307.167,A -85,B 0,C 180,E1 -13830.987,E2 -13830.987} C_VEL
LIN {X 0,Y 347.825,Z 307.155,A -85,B 0,C 180,E1 -13833.607,E2 -13833.607} C_VEL
LIN {X 0,Y 347.783,Z 307.16,A -85,B 0,C 180,E1 -13836.162,E2 -13836.162} C_VEL
LIN {X 0,Y 347.812,Z 307.157,A -85,B 0,C 180,E1 -13839.909,E2 -13839.909} C_VEL
LIN {X 0,Y 347.861,Z 307.15,A -85,B 0,C 180,E1 -13842.359,E2 -13842.359} C_VEL
LIN {X 0,Y 347.892,Z 307.147,A -85,B 0,C 180,E1 -13845.971,E2 -13845.971} C_VEL
LIN {X 0,Y 347.923,Z 307.148,A -85,B 0,C 180,E1 -13849.526,E2 -13849.526} C_VEL
LIN {X 0,Y 348.068,Z 307.127,A -85,B 0,C 180,E1 -13851.875,E2 -13851.875} C_VEL
LIN {X 0,Y 348.061,Z 307.126,A -85,B 0,C 180,E1 -13854.206,E2 -13854.206} C_VEL
LIN {X 0,Y 348.2,Z 307.114,A -85,B 0,C 180,E1 -13857.687,E2 -13857.687} C_VEL
LIN {X 0,Y 348.339,Z 307.094,A -85,B 0,C 180,E1 -13860,E2 -13860} C_VEL
LIN {X 0,Y 348.201,Z 307.109,A -85,B 0,C 180,E1 -13862.314,E2 -13862.314} C_VEL
LIN {X 0,Y 348.065,Z 307.125,A -85,B 0,C 180,E1 -13866.959,E2 -13866.959} C_VEL
LIN {X 0,Y 347.923,Z 307.144,A -85,B 0,C 180,E1 -13870.475,E2 -13870.475} C_VEL
LIN {X 0,Y 347.893,Z 307.152,A -85,B 0,C 180,E1 -13874.15,E2 -13874.15} C_VEL
LIN {X 0,Y 347.886,Z 307.153,A -85,B 0,C 180,E1 -13878.291,E2 -13878.291} C_VEL
LIN {X 0,Y 347.763,Z 307.163,A -85,B 0,C 180,E1 -13881.627,E2 -13881.627} C_VEL
LIN {X 0,Y 347.768,Z 307.162,A -85,B 0,C 180,E1 -13885.112,E2 -13885.112} C_VEL
LIN {X 0,Y 347.735,Z 307.166,A -85,B 0,C 180,E1 -13887.701,E2 -13887.701} C_VEL
LIN {X 0,Y 347.737,Z 307.17,A -85,B 0,C 180,E1 -13890.35,E2 -13890.35} C_VEL
LIN {X 0,Y 347.745,Z 307.165,A -85,B 0,C 180,E1 -13894.045,E2 -13894.045} C_VEL
LIN {X 0,Y 347.755,Z 307.164,A -85,B 0,C 180,E1 -13897.322,E2 -13897.322} C_VEL
LIN {X 0,Y 347.718,Z 307.169,A -85,B 0,C 180,E1 -13900.3,E2 -13900.3} C_VEL
LIN {X 0,Y 347.721,Z 307.169,A -85,B 0,C 180,E1 -13903.409,E2 -13903.409} C_VEL
LIN {X 0,Y 347.722,Z 307.171,A -85,B 0,C 180,E1 -13906.688,E2 -13906.688} C_VEL
LIN {X 0,Y 347.7,Z 307.17,A -85,B 0,C 180,E1 -13910.183,E2 -13910.183} C_VEL
LIN {X 0,Y 347.756,Z 307.165,A -85,B 0,C 180,E1 -13912.68,E2 -13912.68} C_VEL
LIN {X 0,Y 347.748,Z 307.165,A -85,B 0,C 180,E1 -13915.957,E2 -13915.957} C_VEL
LIN {X 0,Y 347.738,Z 307.169,A -85,B 0,C 180,E1 -13919.652,E2 -13919.652} C_VEL
LIN {X 0,Y 347.74,Z 307.17,A -85,B 0,C 180,E1 -13923.601,E2 -13923.601} C_VEL
LIN {X 0,Y 347.76,Z 307.163,A -85,B 0,C 180,E1 -13926.161,E2 -13926.161} C_VEL
LIN {X 0,Y 347.802,Z 307.161,A -85,B 0,C 180,E1 -13929.91,E2 -13929.91} C_VEL
LIN {X 0,Y 347.835,Z 307.158,A -85,B 0,C 180,E1 -13933.569,E2 -13933.569} C_VEL
LIN {X 0,Y 347.89,Z 307.147,A -85,B 0,C 180,E1 -13937.161,E2 -13937.161} C_VEL
LIN {X 0,Y 347.937,Z 307.141,A -85,B 0,C 180,E1 -13940.701,E2 -13940.701} C_VEL
LIN {X 0,Y 348.039,Z 307.132,A -85,B 0,C 180,E1 -13944.206,E2 -13944.206} C_VEL
LIN {X 0,Y 348.156,Z 307.115,A -85,B 0,C 180,E1 -13947.687,E2 -13947.687} C_VEL
LIN {X 0,Y 348.119,Z 307.118,A -85,B 0,C 180,E1 -13951.157,E2 -13951.157} C_VEL
LIN {X 0,Y 348.155,Z 307.119,A -85,B 0,C 180,E1 -13952.314,E2 -13952.314} C_VEL
LIN {X 0,Y 348.059,Z 307.126,A -85,B 0,C 180,E1 -13956.959,E2 -13956.959} C_VEL
LIN {X 0,Y 347.883,Z 307.154,A -85,B 0,C 180,E1 -13960.476,E2 -13960.476} C_VEL
LIN {X 0,Y 347.856,Z 307.153,A -85,B 0,C 180,E1 -13964.119,E2 -13964.119} C_VEL
LIN {X 0,Y 347.798,Z 307.16,A -85,B 0,C 180,E1 -13968.241,E2 -13968.241} C_VEL
LIN {X 0,Y 347.803,Z 307.214,A -85,B 0,C 180,E1 -13972.374,E2 -13972.374} C_VEL
LIN {X 0,Y 349.353,Z 315.117,A -85,B 0,C 180,E1 -13974.673,E2 -13974.673} C_VEL
LIN {X 0,Y 353.518,Z 328.255,A -85,B 0,C 180,E1 -13975.235,E2 -13975.235} C_VEL
LIN {X 0,Y 356.045,Z 342.085,A -85,B 0,C 180,E1 -13975.697,E2 -13975.697} C_VEL
LIN {X 0,Y 354.208,Z 422.834,A -85,B 0,C 180,E1 -13977.492,E2 -13977.492} C_VEL
LIN {X 0,Y 353.54,Z 436.984,A -85,B 0,C 180,E1 -13978.052,E2 -13978.052} C_VEL
LIN {X 0,Y 352.908,Z 449.692,A -85,B 0,C 180,E1 -13978.807,E2 -13978.807} C_VEL
LIN {X 0,Y 351.937,Z 462.201,A -85,B 0,C 180,E1 -13979.806,E2 -13979.806} C_VEL
LIN {X 0,Y 350.955,Z 473.586,A -85,B 0,C 180,E1 -13980.976,E2 -13980.976} C_VEL
LIN {X 0,Y 350.081,Z 483.805,A -85,B 0,C 180,E1 -13982.305,E2 -13982.305} C_VEL
LIN {X 0,Y 349.24,Z 492.074,A -85,B 0,C 180,E1 -13983.61,E2 -13983.61} C_VEL
LIN {X 0,Y 348.111,Z 496.066,A -85,B 0,C 180,E1 -13984.309,E2 -13984.309} C_VEL
LIN {X 0,Y 344.619,Z 502.122,A -85,B 0,C 180,E1 -13985.47,E2 -13985.47} C_VEL
LIN {X 0,Y 341.219,Z 507.603,A -85,B 0,C 180,E1 -13986.729,E2 -13986.729} C_VEL
LIN {X 0,Y 340.249,Z 510.609,A -85,B 0,C 180,E1 -13987.569,E2 -13987.569} C_VEL
LIN {X 0,Y 339.77,Z 516.3,A -85,B 0,C 180,E1 -13989.499,E2 -13989.499} C_VEL
LIN {X 0,Y 339.394,Z 520.728,A -85,B 0,C 180,E1 -13991.502,E2 -13991.502} C_VEL
LIN {X 0,Y 339.027,Z 523.825,A -85,B 0,C 180,E1 -13993.485,E2 -13993.485} C_VEL
LIN {X 0,Y 338.907,Z 525.509,A -85,B 0,C 180,E1 -13995.164,E2 -13995.164} C_VEL
LIN {X 0,Y 338.901,Z 526.375,A -85,B 0,C 180,E1 -13996.815,E2 -13996.815} C_VEL
LIN {X 0,Y 338.922,Z 526.439,A -85,B 0,C 180,E1 -13998.427,E2 -13998.427} C_VEL
LIN {X 0,Y 339.015,Z 525.721,A -85,B 0,C 180,E1 -14000.089,E2 -14000.089} C_VEL
LIN {X 0,Y 339.306,Z 524.015,A -85,B 0,C 180,E1 -14001.915,E2 -14001.915} C_VEL
LIN {X 0,Y 339.733,Z 521.228,A -85,B 0,C 180,E1 -14003.784,E2 -14003.784} C_VEL
LIN {X 0,Y 340.332,Z 517.214,A -85,B 0,C 180,E1 -14005.692,E2 -14005.692} C_VEL
LIN {X 0,Y 341.123,Z 511.776,A -85,B 0,C 180,E1 -14007.641,E2 -14007.641} C_VEL
LIN {X 0,Y 342.158,Z 504.585,A -85,B 0,C 180,E1 -14009.62,E2 -14009.62} C_VEL
LIN {X 0,Y 343.456,Z 496.284,A -85,B 0,C 180,E1 -14011.421,E2 -14011.421} C_VEL
LIN {X 0,Y 344.702,Z 487.091,A -85,B 0,C 180,E1 -14013.022,E2 -14013.022} C_VEL
LIN {X 0,Y 345.996,Z 477.016,A -85,B 0,C 180,E1 -14014.428,E2 -14014.428} C_VEL
LIN {X 0,Y 347.258,Z 466.501,A -85,B 0,C 180,E1 -14015.608,E2 -14015.608} C_VEL
LIN {X 0,Y 348.4,Z 455.381,A -85,B 0,C 180,E1 -14016.6,E2 -14016.6} C_VEL
LIN {X 0,Y 349.457,Z 442.636,A -85,B 0,C 180,E1 -14017.457,E2 -14017.457} C_VEL
LIN {X 0,Y 350.13,Z 430.171,A -85,B 0,C 180,E1 -14018.066,E2 -14018.066} C_VEL
LIN {X 0,Y 350.717,Z 416.657,A -85,B 0,C 180,E1 -14018.471,E2 -14018.471} C_VEL
LIN {X 0,Y 352.857,Z 343.236,A -85,B 0,C 180,E1 -14020.174,E2 -14020.174} C_VEL
LIN {X 0,Y 350.929,Z 334.338,A -85,B 0,C 180,E1 -14020.575,E2 -14020.575} C_VEL
LIN {X 0,Y 344.317,Z 318.999,A -85,B 0,C 180,E1 -14021.594,E2 -14021.594} C_VEL
LIN {X 0,Y 342.814,Z 315.673,A -85,B 0,C 180,E1 -14021.859,E2 -14021.859} C_VEL
LIN {X 0,Y 340.792,Z 308.041,A -85,B 0,C 180,E1 -14023.988,E2 -14023.988} C_VEL
LIN {X 0,Y 340.847,Z 308.03,A -85,B 0,C 180,E1 -14026.89,E2 -14026.89} C_VEL
LIN {X 0,Y 340.931,Z 308.018,A -85,B 0,C 180,E1 -14030.507,E2 -14030.507} C_VEL
LIN {X 0,Y 341.077,Z 308,A -85,B 0,C 180,E1 -14032.898,E2 -14032.898} C_VEL
LIN {X 0,Y 341.17,Z 307.988,A -85,B 0,C 180,E1 -14037.638,E2 -14037.638} C_VEL
LIN {X 0,Y 341.278,Z 307.974,A -85,B 0,C 180,E1 -14040,E2 -14040} C_VEL
LIN {X 0,Y 341.17,Z 307.988,A -85,B 0,C 180,E1 -14042.361,E2 -14042.361} C_VEL
LIN {X 0,Y 341.02,Z 307.998,A -85,B 0,C 180,E1 -14047.103,E2 -14047.103} C_VEL
LIN {X 0,Y 340.873,Z 308.02,A -85,B 0,C 180,E1 -14050.694,E2 -14050.694} C_VEL
LIN {X 0,Y 340.865,Z 308.02,A -85,B 0,C 180,E1 -14054.325,E2 -14054.325} C_VEL
LIN {X 0,Y 340.787,Z 308.033,A -85,B 0,C 180,E1 -14058.44,E2 -14058.44} C_VEL
LIN {X 0,Y 340.719,Z 308.038,A -85,B 0,C 180,E1 -14061.841,E2 -14061.841} C_VEL
LIN {X 0,Y 340.774,Z 308.033,A -85,B 0,C 180,E1 -14065.664,E2 -14065.664} C_VEL
LIN {X 0,Y 340.73,Z 308.033,A -85,B 0,C 180,E1 -14068.32,E2 -14068.32} C_VEL
LIN {X 0,Y 340.699,Z 308.04,A -85,B 0,C 180,E1 -14071.044,E2 -14071.044} C_VEL
LIN {X 0,Y 340.719,Z 308.04,A -85,B 0,C 180,E1 -14075.279,E2 -14075.279} C_VEL
LIN {X 0,Y 340.711,Z 308.04,A -85,B 0,C 180,E1 -14078.386,E2 -14078.386} C_VEL
LIN {X 0,Y 340.701,Z 308.047,A -85,B 0,C 180,E1 -14082.045,E2 -14082.045} C_VEL
LIN {X 0,Y 340.654,Z 308.05,A -85,B 0,C 180,E1 -14086.227,E2 -14086.227} C_VEL
LIN {X 0,Y 340.69,Z 308.047,A -85,B 0,C 180,E1 -14089.753,E2 -14089.753} C_VEL
LIN {X 0,Y 340.707,Z 308.049,A -85,B 0,C 180,E1 -14093.258,E2 -14093.258} C_VEL
LIN {X 0,Y 340.694,Z 308.054,A -85,B 0,C 180,E1 -14096.153,E2 -14096.153} C_VEL
LIN {X 0,Y 340.692,Z 308.095,A -85,B 0,C 180,E1 -14097.755,E2 -14097.755} C_VEL
LIN {X 0,Y 343.526,Z 319.041,A -85,B 0,C 180,E1 -14100.861,E2 -14100.861} C_VEL
LIN {X 0,Y 345.684,Z 329.97,A -85,B 0,C 180,E1 -14103.749,E2 -14103.749} C_VEL
LIN {X 0,Y 345.203,Z 336.748,A -85,B 0,C 180,E1 -14105.331,E2 -14105.331} C_VEL
LIN {X 0,Y 345.136,Z 337.255,A -85,B 0,C 180,E1 -14105.446,E2 -14105.446} C_VEL
LIN {X 0,Y 349.5,Z 358.902,A -85,B 0,C 180,E1 -14106.416,E2 -14106.416} C_VEL
LIN {X 0,Y 352.113,Z 377.333,A -85,B 0,C 180,E1 -14107.117,E2 -14107.117} C_VEL
LIN {X 0,Y 350.054,Z 448.038,A -85,B 0,C 180,E1 -14108.778,E2 -14108.778} C_VEL
LIN {X 0,Y 349.133,Z 461.775,A -85,B 0,C 180,E1 -14109.335,E2 -14109.335} C_VEL
LIN {X 0,Y 348.047,Z 474.19,A -85,B 0,C 180,E1 -14110.077,E2 -14110.077} C_VEL
LIN {X 0,Y 346.847,Z 484.999,A -85,B 0,C 180,E1 -14110.929,E2 -14110.929} C_VEL
LIN {X 0,Y 345.444,Z 496.426,A -85,B 0,C 180,E1 -14112.078,E2 -14112.078} C_VEL
LIN {X 0,Y 344.116,Z 506.793,A -85,B 0,C 180,E1 -14113.385,E2 -14113.385} C_VEL
LIN {X 0,Y 342.838,Z 516.143,A -85,B 0,C 180,E1 -14114.848,E2 -14114.848} C_VEL
LIN {X 0,Y 341.813,Z 523.876,A -85,B 0,C 180,E1 -14116.322,E2 -14116.322} C_VEL
LIN {X 0,Y 340.68,Z 531.492,A -85,B 0,C 180,E1 -14118.094,E2 -14118.094} C_VEL
LIN {X 0,Y 339.964,Z 537.641,A -85,B 0,C 180,E1 -14119.879,E2 -14119.879} C_VEL
LIN {X 0,Y 339.51,Z 542.521,A -85,B 0,C 180,E1 -14121.668,E2 -14121.668} C_VEL
LIN {X 0,Y 339.196,Z 546.267,A -85,B 0,C 180,E1 -14123.456,E2 -14123.456} C_VEL
LIN {X 0,Y 339.075,Z 548.984,A -85,B 0,C 180,E1 -14125.244,E2 -14125.244} C_VEL
LIN {X 0,Y 339.072,Z 550.279,A -85,B 0,C 180,E1 -14126.434,E2 -14126.434} C_VEL
LIN {X 0,Y 339.024,Z 551.127,A -85,B 0,C 180,E1 -14127.623,E2 -14127.623} C_VEL
LIN {X 0,Y 339.072,Z 551.555,A -85,B 0,C 180,E1 -14128.812,E2 -14128.812} C_VEL
LIN {X 0,Y 339.139,Z 551.587,A -85,B 0,C 180,E1 -14129.999,E2 -14129.999} C_VEL
LIN {X 0,Y 339.089,Z 551.215,A -85,B 0,C 180,E1 -14131.187,E2 -14131.187} C_VEL
LIN {X 0,Y 339.029,Z 550.394,A -85,B 0,C 180,E1 -14132.375,E2 -14132.375} C_VEL
LIN {X 0,Y 339.076,Z 549.149,A -85,B 0,C 180,E1 -14133.564,E2 -14133.564} C_VEL
LIN {X 0,Y 339.094,Z 547.482,A -85,B 0,C 180,E1 -14134.755,E2 -14134.755} C_VEL
LIN {X 0,Y 339.192,Z 544.099,A -85,B 0,C 180,E1 -14136.543,E2 -14136.543} C_VEL
LIN {X 0,Y 339.454,Z 539.602,A -85,B 0,C 180,E1 -14138.332,E2 -14138.332} C_VEL
LIN {X 0,Y 339.867,Z 533.86,A -85,B 0,C 180,E1 -14140.123,E2 -14140.123} C_VEL
LIN {X 0,Y 340.541,Z 526.631,A -85,B 0,C 180,E1 -14141.909,E2 -14141.909} C_VEL
LIN {X 0,Y 341.46,Z 517.604,A -85,B 0,C 180,E1 -14143.691,E2 -14143.691} C_VEL
LIN {X 0,Y 342.389,Z 508.729,A -85,B 0,C 180,E1 -14145.11,E2 -14145.11} C_VEL
LIN {X 0,Y 343.373,Z 498.012,A -85,B 0,C 180,E1 -14146.497,E2 -14146.497} C_VEL
LIN {X 0,Y 344.519,Z 486.604,A -85,B 0,C 180,E1 -14147.664,E2 -14147.664} C_VEL
LIN {X 0,Y 345.553,Z 474.806,A -85,B 0,C 180,E1 -14148.605,E2 -14148.605} C_VEL
LIN {X 0,Y 346.424,Z 461.919,A -85,B 0,C 180,E1 -14149.363,E2 -14149.363} C_VEL
LIN {X 0,Y 347.196,Z 448.483,A -85,B 0,C 180,E1 -14149.896,E2 -14149.896} C_VEL
LIN {X 0,Y 348.671,Z 375.157,A -85,B 0,C 180,E1 -14151.579,E2 -14151.579} C_VEL
LIN {X 0,Y 343.546,Z 339.607,A -85,B 0,C 180,E1 -14152.735,E2 -14152.735} C_VEL
LIN {X 0,Y 344.687,Z 328.699,A -85,B 0,C 180,E1 -14155.351,E2 -14155.351} C_VEL
LIN {X 0,Y 343.665,Z 322.066,A -85,B 0,C 180,E1 -14157.065,E2 -14157.065} C_VEL
LIN {X 0,Y 341.313,Z 310.651,A -85,B 0,C 180,E1 -14160.137,E2 -14160.137} C_VEL
LIN {X 0,Y 340.744,Z 308.037,A -85,B 0,C 180,E1 -14160.909,E2 -14160.909} C_VEL
LIN {X 0,Y 340.715,Z 308.04,A -85,B 0,C 180,E1 -14165.278,E2 -14165.278} C_VEL
LIN {X 0,Y 340.707,Z 308.047,A -85,B 0,C 180,E1 -14168.385,E2 -14168.385} C_VEL
LIN {X 0,Y 340.695,Z 308.045,A -85,B 0,C 180,E1 -14172.045,E2 -14172.045} C_VEL
LIN {X 0,Y 340.648,Z 308.052,A -85,B 0,C 180,E1 -14176.226,E2 -14176.226} C_VEL
LIN {X 0,Y 340.684,Z 308.044,A -85,B 0,C 180,E1 -14179.752,E2 -14179.752} C_VEL
LIN {X 0,Y 340.703,Z 308.043,A -85,B 0,C 180,E1 -14183.258,E2 -14183.258} C_VEL
LIN {X 0,Y 340.687,Z 308.044,A -85,B 0,C 180,E1 -14186.153,E2 -14186.153} C_VEL
LIN {X 0,Y 340.736,Z 308.039,A -85,B 0,C 180,E1 -14190.329,E2 -14190.329} C_VEL
LIN {X 0,Y 340.798,Z 308.036,A -85,B 0,C 180,E1 -14193.02,E2 -14193.02} C_VEL
LIN {X 0,Y 340.75,Z 308.037,A -85,B 0,C 180,E1 -14195.638,E2 -14195.638} C_VEL
LIN {X 0,Y 340.743,Z 308.04,A -85,B 0,C 180,E1 -14199.474,E2 -14199.474} C_VEL
LIN {X 0,Y 340.852,Z 308.023,A -85,B 0,C 180,E1 -14201.984,E2 -14201.984} C_VEL
LIN {X 0,Y 340.863,Z 308.024,A -85,B 0,C 180,E1 -14205.705,E2 -14205.705} C_VEL
LIN {X 0,Y 340.865,Z 308.027,A -85,B 0,C 180,E1 -14209.306,E2 -14209.306} C_VEL
LIN {X 0,Y 341.07,Z 307.997,A -85,B 0,C 180,E1 -14212.898,E2 -14212.898} C_VEL
LIN {X 0,Y 341.162,Z 307.991,A -85,B 0,C 180,E1 -14217.639,E2 -14217.639} C_VEL
LIN {X 0,Y 341.289,Z 307.972,A -85,B 0,C 180,E1 -14220,E2 -14220} C_VEL
LIN {X 0,Y 341.162,Z 307.986,A -85,B 0,C 180,E1 -14222.362,E2 -14222.362} C_VEL
LIN {X 0,Y 341.012,Z 308.003,A -85,B 0,C 180,E1 -14227.103,E2 -14227.103} C_VEL
LIN {X 0,Y 340.865,Z 308.022,A -85,B 0,C 180,E1 -14230.694,E2 -14230.694} C_VEL
LIN {X 0,Y 340.858,Z 308.027,A -85,B 0,C 180,E1 -14234.325,E2 -14234.325} C_VEL
LIN {X 0,Y 340.833,Z 308.029,A -85,B 0,C 180,E1 -14238.467,E2 -14238.467} C_VEL
LIN {X 0,Y 340.713,Z 308.042,A -85,B 0,C 180,E1 -14241.842,E2 -14241.842} C_VEL
LIN {X 0,Y 340.72,Z 308.04,A -85,B 0,C 180,E1 -14245.669,E2 -14245.669} C_VEL
LIN {X 0,Y 340.704,Z 308.042,A -85,B 0,C 180,E1 -14249.675,E2 -14249.675} C_VEL
LIN {X 0,Y 340.682,Z 308.049,A -85,B 0,C 180,E1 -14252.437,E2 -14252.437} C_VEL
LIN {X 0,Y 340.715,Z 308.041,A -85,B 0,C 180,E1 -14255.28,E2 -14255.28} C_VEL
LIN {X 0,Y 340.692,Z 308.046,A -85,B 0,C 180,E1 -14258.384,E2 -14258.384} C_VEL
LIN {X 0,Y 340.696,Z 308.043,A -85,B 0,C 180,E1 -14262.046,E2 -14262.046} C_VEL
LIN {X 0,Y 340.649,Z 308.049,A -85,B 0,C 180,E1 -14266.228,E2 -14266.228} C_VEL
LIN {X 0,Y 340.67,Z 308.049,A -85,B 0,C 180,E1 -14268.689,E2 -14268.689} C_VEL
LIN {X 0,Y 340.718,Z 308.041,A -85,B 0,C 180,E1 -14271.772,E2 -14271.772} C_VEL
LIN {X 0,Y 340.723,Z 308.042,A -85,B 0,C 180,E1 -14275.597,E2 -14275.597} C_VEL
LIN {X 0,Y 340.693,Z 308.046,A -85,B 0,C 180,E1 -14278.956,E2 -14278.956} C_VEL
LIN {X 0,Y 340.712,Z 308.043,A -85,B 0,C 180,E1 -14283.013,E2 -14283.013} C_VEL
LIN {X 0,Y 340.746,Z 308.041,A -85,B 0,C 180,E1 -14285.639,E2 -14285.639} C_VEL
LIN {X 0,Y 340.733,Z 308.043,A -85,B 0,C 180,E1 -14289.474,E2 -14289.474} C_VEL
LIN {X 0,Y 340.795,Z 308.034,A -85,B 0,C 180,E1 -14291.982,E2 -14291.982} C_VEL
LIN {X 0,Y 340.873,Z 308.026,A -85,B 0,C 180,E1 -14295.706,E2 -14295.706} C_VEL
LIN {X 0,Y 340.846,Z 308.025,A -85,B 0,C 180,E1 -14299.306,E2 -14299.306} C_VEL
LIN {X 0,Y 341.003,Z 308.004,A -85,B 0,C 180,E1 -14302.897,E2 -14302.897} C_VEL
LIN {X 0,Y 340.806,Z 308.029,A -85,B 0,C 180,E1 -14305.269,E2 -14305.269} C_VEL
LIN {X 0,Y 341.097,Z 307.995,A -85,B 0,C 180,E1 -14307.639,E2 -14307.639} C_VEL
LIN {X 0,Y 341.09,Z 307.993,A -85,B 0,C 180,E1 -14311.181,E2 -14311.181} C_VEL
LIN {X 0,Y 341.095,Z 307.998,A -85,B 0,C 180,E1 -14312.362,E2 -14312.362} C_VEL
LIN {X 0,Y 341.015,Z 308.005,A -85,B 0,C 180,E1 -14315.915,E2 -14315.915} C_VEL
LIN {X 0,Y 340.968,Z 308.015,A -85,B 0,C 180,E1 -14318.357,E2 -14318.357} C_VEL
LIN {X 0,Y 340.836,Z 308.026,A -85,B 0,C 180,E1 -14321.9,E2 -14321.9} C_VEL
LIN {X 0,Y 340.747,Z 308.036,A -85,B 0,C 180,E1 -14325.554,E2 -14325.554} C_VEL
LIN {X 0,Y 340.76,Z 308.038,A -85,B 0,C 180,E1 -14328.425,E2 -14328.425} C_VEL
LIN {X 0,Y 340.781,Z 308.168,A -85,B 0,C 180,E1 -14332.121,E2 -14332.121} C_VEL
LIN {X 0,Y 342.266,Z 315.645,A -85,B 0,C 180,E1 -14334.288,E2 -14334.288} C_VEL
LIN {X 0,Y 346.884,Z 329.734,A -85,B 0,C 180,E1 -14334.901,E2 -14334.901} C_VEL
LIN {X 0,Y 349.279,Z 342.452,A -85,B 0,C 180,E1 -14335.341,E2 -14335.341} C_VEL
LIN {X 0,Y 347.401,Z 423.024,A -85,B 0,C 180,E1 -14337.173,E2 -14337.173} C_VEL
LIN {X 0,Y 346.725,Z 437.128,A -85,B 0,C 180,E1 -14337.74,E2 -14337.74} C_VEL
LIN {X 0,Y 346.048,Z 449.856,A -85,B 0,C 180,E1 -14338.508,E2 -14338.508} C_VEL
LIN {X 0,Y 345.079,Z 462.235,A -85,B 0,C 180,E1 -14339.513,E2 -14339.513} C_VEL
LIN {X 0,Y 344.037,Z 473.721,A -85,B 0,C 180,E1 -14340.711,E2 -14340.711} C_VEL
LIN {X 0,Y 343.165,Z 483.582,A -85,B 0,C 180,E1 -14342.009,E2 -14342.009} C_VEL
LIN {X 0,Y 342.261,Z 492.43,A -85,B 0,C 180,E1 -14343.429,E2 -14343.429} C_VEL
LIN {X 0,Y 341.209,Z 501.502,A -85,B 0,C 180,E1 -14345.221,E2 -14345.221} C_VEL
LIN {X 0,Y 340.521,Z 507.802,A -85,B 0,C 180,E1 -14346.765,E2 -14346.765} C_VEL
LIN {X 0,Y 340.249,Z 510.609,A -85,B 0,C 180,E1 -14347.569,E2 -14347.569} C_VEL
LIN {X 0,Y 339.317,Z 513.414,A -85,B 0,C 180,E1 -14348.435,E2 -14348.435} C_VEL
LIN {X 0,Y 334.713,Z 518.904,A -85,B 0,C 180,E1 -14350.46,E2 -14350.46} C_VEL
LIN {X 0,Y 332.546,Z 521.436,A -85,B 0,C 180,E1 -14351.699,E2 -14351.699} C_VEL
LIN {X 0,Y 332.112,Z 522.516,A -85,B 0,C 180,E1 -14352.351,E2 -14352.351} C_VEL
LIN {X 0,Y 331.84,Z 525.039,A -85,B 0,C 180,E1 -14354.34,E2 -14354.34} C_VEL
LIN {X 0,Y 331.778,Z 526.322,A -85,B 0,C 180,E1 -14356.073,E2 -14356.073} C_VEL
LIN {X 0,Y 331.8,Z 526.78,A -85,B 0,C 180,E1 -14357.847,E2 -14357.847} C_VEL
LIN {X 0,Y 331.896,Z 526.337,A -85,B 0,C 180,E1 -14359.669,E2 -14359.669} C_VEL
LIN {X 0,Y 332.149,Z 524.928,A -85,B 0,C 180,E1 -14361.526,E2 -14361.526} C_VEL
LIN {X 0,Y 332.664,Z 521.964,A -85,B 0,C 180,E1 -14363.733,E2 -14363.733} C_VEL
LIN {X 0,Y 333.129,Z 518.855,A -85,B 0,C 180,E1 -14365.365,E2 -14365.365} C_VEL
LIN {X 0,Y 333.899,Z 513.835,A -85,B 0,C 180,E1 -14367.345,E2 -14367.345} C_VEL
LIN {X 0,Y 334.942,Z 507.228,A -85,B 0,C 180,E1 -14369.35,E2 -14369.35} C_VEL
LIN {X 0,Y 336.262,Z 499.163,A -85,B 0,C 180,E1 -14371.268,E2 -14371.268} C_VEL
LIN {X 0,Y 337.559,Z 490.379,A -85,B 0,C 180,E1 -14372.927,E2 -14372.927} C_VEL
LIN {X 0,Y 338.838,Z 481.179,A -85,B 0,C 180,E1 -14374.34,E2 -14374.34} C_VEL
LIN {X 0,Y 340.182,Z 471.107,A -85,B 0,C 180,E1 -14375.594,E2 -14375.594} C_VEL
LIN {X 0,Y 341.397,Z 460.546,A -85,B 0,C 180,E1 -14376.654,E2 -14376.654} C_VEL
LIN {X 0,Y 342.582,Z 448.269,A -85,B 0,C 180,E1 -14377.605,E2 -14377.605} C_VEL
LIN {X 0,Y 343.427,Z 435.354,A -85,B 0,C 180,E1 -14378.353,E2 -14378.353} C_VEL
LIN {X 0,Y 344.147,Z 423.205,A -85,B 0,C 180,E1 -14378.813,E2 -14378.813} C_VEL
LIN {X 0,Y 346.52,Z 344.076,A -85,B 0,C 180,E1 -14380.709,E2 -14380.709} C_VEL
LIN {X 0,Y 344.882,Z 336.762,A -85,B 0,C 180,E1 -14381.055,E2 -14381.055} C_VEL
LIN {X 0,Y 338.744,Z 322.577,A -85,B 0,C 180,E1 -14382.043,E2 -14382.043} C_VEL
LIN {X 0,Y 335.677,Z 316.041,A -85,B 0,C 180,E1 -14382.563,E2 -14382.563} C_VEL
LIN {X 0,Y 333.8,Z 308.912,A -85,B 0,C 180,E1 -14384.663,E2 -14384.663} C_VEL
LIN {X 0,Y 333.794,Z 308.908,A -85,B 0,C 180,E1 -14387.845,E2 -14387.845} C_VEL
LIN {X 0,Y 334.001,Z 308.88,A -85,B 0,C 180,E1 -14391.53,E2 -14391.53} C_VEL
LIN {X 0,Y 334.022,Z 308.878,A -85,B 0,C 180,E1 -14393.961,E2 -14393.961} C_VEL
LIN {X 0,Y 334.107,Z 308.868,A -85,B 0,C 180,E1 -14397.589,E2 -14397.589} C_VEL
LIN {X 0,Y 334.23,Z 308.852,A -85,B 0,C 180,E1 -14400,E2 -14400} C_VEL
LIN {X 0,Y 334.107,Z 308.868,A -85,B 0,C 180,E1 -14402.411,E2 -14402.411} C_VEL
LIN {X 0,Y 334.003,Z 308.878,A -85,B 0,C 180,E1 -14406.039,E2 -14406.039} C_VEL
LIN {X 0,Y 333.851,Z 308.895,A -85,B 0,C 180,E1 -14409.695,E2 -14409.695} C_VEL
LIN {X 0,Y 333.799,Z 308.898,A -85,B 0,C 180,E1 -14413.391,E2 -14413.391} C_VEL
LIN {X 0,Y 333.72,Z 308.907,A -85,B 0,C 180,E1 -14417.147,E2 -14417.147} C_VEL
LIN {X 0,Y 333.687,Z 308.918,A -85,B 0,C 180,E1 -14419.693,E2 -14419.693} C_VEL
LIN {X 0,Y 333.672,Z 308.917,A -85,B 0,C 180,E1 -14423.59,E2 -14423.59} C_VEL
LIN {X 0,Y 333.737,Z 308.911,A -85,B 0,C 180,E1 -14426.246,E2 -14426.246} C_VEL
LIN {X 0,Y 333.692,Z 308.915,A -85,B 0,C 180,E1 -14428.974,E2 -14428.974} C_VEL
LIN {X 0,Y 333.645,Z 308.922,A -85,B 0,C 180,E1 -14432.587,E2 -14432.587} C_VEL
LIN {X 0,Y 333.678,Z 308.92,A -85,B 0,C 180,E1 -14436.139,E2 -14436.139} C_VEL
LIN {X 0,Y 333.648,Z 308.926,A -85,B 0,C 180,E1 -14439.192,E2 -14439.192} C_VEL
LIN {X 0,Y 333.634,Z 308.927,A -85,B 0,C 180,E1 -14442.5,E2 -14442.5} C_VEL
LIN {X 0,Y 333.598,Z 308.929,A -85,B 0,C 180,E1 -14445.955,E2 -14445.955} C_VEL
LIN {X 0,Y 333.649,Z 308.927,A -85,B 0,C 180,E1 -14449.315,E2 -14449.315} C_VEL
LIN {X 0,Y 333.667,Z 308.927,A -85,B 0,C 180,E1 -14453.167,E2 -14453.167} C_VEL
LIN {X 0,Y 333.676,Z 308.928,A -85,B 0,C 180,E1 -14455.341,E2 -14455.341} C_VEL
LIN {X 0,Y 333.647,Z 309.074,A -85,B 0,C 180,E1 -14457.158,E2 -14457.158} C_VEL
LIN {X 0,Y 336.4,Z 319.594,A -85,B 0,C 180,E1 -14460.252,E2 -14460.252} C_VEL
LIN {X 0,Y 338.373,Z 328.876,A -85,B 0,C 180,E1 -14462.81,E2 -14462.81} C_VEL
LIN {X 0,Y 338.941,Z 333.236,A -85,B 0,C 180,E1 -14463.941,E2 -14463.941} C_VEL
LIN {X 0,Y 338.531,Z 337.069,A -85,B 0,C 180,E1 -14464.811,E2 -14464.811} C_VEL
LIN {X 0,Y 342.912,Z 358.237,A -85,B 0,C 180,E1 -14465.813,E2 -14465.813} C_VEL
LIN {X 0,Y 345.797,Z 377.932,A -85,B 0,C 180,E1 -14466.595,E2 -14466.595} C_VEL
LIN {X 0,Y 343.64,Z 446.875,A -85,B 0,C 180,E1 -14468.245,E2 -14468.245} C_VEL
LIN {X 0,Y 342.72,Z 460.784,A -85,B 0,C 180,E1 -14468.812,E2 -14468.812} C_VEL
LIN {X 0,Y 341.64,Z 472.879,A -85,B 0,C 180,E1 -14469.53,E2 -14469.53} C_VEL
LIN {X 0,Y 340.173,Z 485.486,A -85,B 0,C 180,E1 -14470.54,E2 -14470.54} C_VEL
LIN {X 0,Y 338.726,Z 496.779,A -85,B 0,C 180,E1 -14471.71,E2 -14471.71} C_VEL
LIN {X 0,Y 337.315,Z 507.021,A -85,B 0,C 180,E1 -14473.04,E2 -14473.04} C_VEL
LIN {X 0,Y 335.987,Z 516.272,A -85,B 0,C 180,E1 -14474.532,E2 -14474.532} C_VEL
LIN {X 0,Y 334.694,Z 525.321,A -85,B 0,C 180,E1 -14476.335,E2 -14476.335} C_VEL
LIN {X 0,Y 333.555,Z 532.63,A -85,B 0,C 180,E1 -14478.145,E2 -14478.145} C_VEL
LIN {X 0,Y 332.954,Z 537.578,A -85,B 0,C 180,E1 -14479.663,E2 -14479.663} C_VEL
LIN {X 0,Y 332.458,Z 542.405,A -85,B 0,C 180,E1 -14481.49,E2 -14481.49} C_VEL
LIN {X 0,Y 332.118,Z 546.114,A -85,B 0,C 180,E1 -14483.316,E2 -14483.316} C_VEL
LIN {X 0,Y 331.982,Z 548.796,A -85,B 0,C 180,E1 -14485.142,E2 -14485.142} C_VEL
LIN {X 0,Y 331.997,Z 550.07,A -85,B 0,C 180,E1 -14486.358,E2 -14486.358} C_VEL
LIN {X 0,Y 331.94,Z 550.885,A -85,B 0,C 180,E1 -14487.572,E2 -14487.572} C_VEL
LIN {X 0,Y 331.974,Z 551.295,A -85,B 0,C 180,E1 -14488.786,E2 -14488.786} C_VEL
LIN {X 0,Y 332.044,Z 551.309,A -85,B 0,C 180,E1 -14489.999,E2 -14489.999} C_VEL
LIN {X 0,Y 331.991,Z 550.912,A -85,B 0,C 180,E1 -14491.212,E2 -14491.212} C_VEL
LIN {X 0,Y 331.944,Z 550.058,A -85,B 0,C 180,E1 -14492.426,E2 -14492.426} C_VEL
LIN {X 0,Y 332.002,Z 548.792,A -85,B 0,C 180,E1 -14493.64,E2 -14493.64} C_VEL
LIN {X 0,Y 332.028,Z 545.429,A -85,B 0,C 180,E1 -14495.821,E2 -14495.821} C_VEL
LIN {X 0,Y 332.305,Z 540.772,A -85,B 0,C 180,E1 -14497.901,E2 -14497.901} C_VEL
LIN {X 0,Y 332.753,Z 534.357,A -85,B 0,C 180,E1 -14500.034,E2 -14500.034} C_VEL
LIN {X 0,Y 333.389,Z 527.35,A -85,B 0,C 180,E1 -14501.86,E2 -14501.86} C_VEL
LIN {X 0,Y 334.204,Z 520.186,A -85,B 0,C 180,E1 -14503.374,E2 -14503.374} C_VEL
LIN {X 0,Y 335.231,Z 510.711,A -85,B 0,C 180,E1 -14505.005,E2 -14505.005} C_VEL
LIN {X 0,Y 336.281,Z 499.583,A -85,B 0,C 180,E1 -14506.543,E2 -14506.543} C_VEL
LIN {X 0,Y 337.367,Z 488.645,A -85,B 0,C 180,E1 -14507.737,E2 -14507.737} C_VEL
LIN {X 0,Y 338.523,Z 476.435,A -85,B 0,C 180,E1 -14508.77,E2 -14508.77} C_VEL
LIN {X 0,Y 339.496,Z 463.739,A -85,B 0,C 180,E1 -14509.578,E2 -14509.578} C_VEL
LIN {X 0,Y 340.287,Z 450.21,A -85,B 0,C 180,E1 -14510.16,E2 -14510.16} C_VEL
LIN {X 0,Y 340.77,Z 429.713,A -85,B 0,C 180,E1 -14510.681,E2 -14510.681} C_VEL
LIN {X 0,Y 341.883,Z 375.575,A -85,B 0,C 180,E1 -14511.933,E2 -14511.933} C_VEL
LIN {X 0,Y 336.668,Z 339.326,A -85,B 0,C 180,E1 -14513.151,E2 -14513.151} C_VEL
LIN {X 0,Y 337.729,Z 329.431,A -85,B 0,C 180,E1 -14515.581,E2 -14515.581} C_VEL
LIN {X 0,Y 336.119,Z 320.346,A -85,B 0,C 180,E1 -14518.001,E2 -14518.001} C_VEL
LIN {X 0,Y 333.691,Z 308.915,A -85,B 0,C 180,E1 -14521.239,E2 -14521.239} C_VEL
LIN {X 0,Y 333.683,Z 308.918,A -85,B 0,C 180,E1 -14524.773,E2 -14524.773} C_VEL
LIN {X 0,Y 333.649,Z 308.921,A -85,B 0,C 180,E1 -14527.65,E2 -14527.65} C_VEL
LIN {X 0,Y 333.643,Z 308.924,A -85,B 0,C 180,E1 -14530.767,E2 -14530.767} C_VEL
LIN {X 0,Y 333.59,Z 308.932,A -85,B 0,C 180,E1 -14534.25,E2 -14534.25} C_VEL
LIN {X 0,Y 333.638,Z 308.922,A -85,B 0,C 180,E1 -14537.618,E2 -14537.618} C_VEL
LIN {X 0,Y 333.65,Z 308.922,A -85,B 0,C 180,E1 -14541.201,E2 -14541.201} C_VEL
LIN {X 0,Y 333.673,Z 308.918,A -85,B 0,C 180,E1 -14543.861,E2 -14543.861} C_VEL
LIN {X 0,Y 333.638,Z 308.923,A -85,B 0,C 180,E1 -14547.413,E2 -14547.413} C_VEL
LIN {X 0,Y 333.685,Z 308.921,A -85,B 0,C 180,E1 -14551.026,E2 -14551.026} C_VEL
LIN {X 0,Y 333.73,Z 308.911,A -85,B 0,C 180,E1 -14553.753,E2 -14553.753} C_VEL
LIN {X 0,Y 333.714,Z 308.913,A -85,B 0,C 180,E1 -14557.914,E2 -14557.914} C_VEL
LIN {X 0,Y 333.789,Z 308.906,A -85,B 0,C 180,E1 -14561.589,E2 -14561.589} C_VEL
LIN {X 0,Y 333.803,Z 308.905,A -85,B 0,C 180,E1 -14565.576,E2 -14565.576} C_VEL
LIN {X 0,Y 333.828,Z 308.901,A -85,B 0,C 180,E1 -14569.078,E2 -14569.078} C_VEL
LIN {X 0,Y 334.02,Z 308.875,A -85,B 0,C 180,E1 -14572.748,E2 -14572.748} C_VEL
LIN {X 0,Y 333.804,Z 308.903,A -85,B 0,C 180,E1 -14575.169,E2 -14575.169} C_VEL
LIN {X 0,Y 334.099,Z 308.87,A -85,B 0,C 180,E1 -14577.589,E2 -14577.589} C_VEL
LIN {X 0,Y 334.24,Z 308.85,A -85,B 0,C 180,E1 -14580,E2 -14580} C_VEL
LIN {X 0,Y 334.1,Z 308.865,A -85,B 0,C 180,E1 -14582.412,E2 -14582.412} C_VEL
LIN {X 0,Y 333.966,Z 308.882,A -85,B 0,C 180,E1 -14586.497,E2 -14586.497} C_VEL
LIN {X 0,Y 333.844,Z 308.899,A -85,B 0,C 180,E1 -14589.696,E2 -14589.696} C_VEL
LIN {X 0,Y 333.792,Z 308.903,A -85,B 0,C 180,E1 -14593.392,E2 -14593.392} C_VEL
LIN {X 0,Y 333.741,Z 308.909,A -85,B 0,C 180,E1 -14597.147,E2 -14597.147} C_VEL
LIN {X 0,Y 333.728,Z 308.912,A -85,B 0,C 180,E1 -14599.691,E2 -14599.691} C_VEL
LIN {X 0,Y 333.655,Z 308.92,A -85,B 0,C 180,E1 -14603.592,E2 -14603.592} C_VEL
LIN {X 0,Y 333.656,Z 308.924,A -85,B 0,C 180,E1 -14606.254,E2 -14606.254} C_VEL
LIN {X 0,Y 333.658,Z 308.923,A -85,B 0,C 180,E1 -14610.279,E2 -14610.279} C_VEL
LIN {X 0,Y 333.633,Z 308.924,A -85,B 0,C 180,E1 -14613.209,E2 -14613.209} C_VEL
LIN {X 0,Y 333.672,Z 308.919,A -85,B 0,C 180,E1 -14616.14,E2 -14616.14} C_VEL
LIN {X 0,Y 333.63,Z 308.925,A -85,B 0,C 180,E1 -14619.195,E2 -14619.195} C_VEL
LIN {X 0,Y 333.63,Z 308.925,A -85,B 0,C 180,E1 -14622.501,E2 -14622.501} C_VEL
LIN {X 0,Y 333.594,Z 308.927,A -85,B 0,C 180,E1 -14625.956,E2 -14625.956} C_VEL
LIN {X 0,Y 333.601,Z 308.93,A -85,B 0,C 180,E1 -14629.326,E2 -14629.326} C_VEL
LIN {X 0,Y 333.662,Z 308.925,A -85,B 0,C 180,E1 -14633.169,E2 -14633.169} C_VEL
LIN {X 0,Y 333.674,Z 308.923,A -85,B 0,C 180,E1 -14635.342,E2 -14635.342} C_VEL
LIN {X 0,Y 333.629,Z 308.923,A -85,B 0,C 180,E1 -14638.223,E2 -14638.223} C_VEL
LIN {X 0,Y 333.652,Z 308.923,A -85,B 0,C 180,E1 -14641.023,E2 -14641.023} C_VEL
LIN {X 0,Y 333.697,Z 308.917,A -85,B 0,C 180,E1 -14645.089,E2 -14645.089} C_VEL
LIN {X 0,Y 333.666,Z 308.919,A -85,B 0,C 180,E1 -14649.019,E2 -14649.019} C_VEL
LIN {X 0,Y 333.743,Z 308.914,A -85,B 0,C 180,E1 -14651.587,E2 -14651.587} C_VEL
LIN {X 0,Y 333.811,Z 308.904,A -85,B 0,C 180,E1 -14655.578,E2 -14655.578} C_VEL
LIN {X 0,Y 333.817,Z 308.9,A -85,B 0,C 180,E1 -14659.078,E2 -14659.078} C_VEL
LIN {X 0,Y 333.959,Z 308.882,A -85,B 0,C 180,E1 -14662.747,E2 -14662.747} C_VEL
LIN {X 0,Y 333.774,Z 308.905,A -85,B 0,C 180,E1 -14665.169,E2 -14665.169} C_VEL
LIN {X 0,Y 334.04,Z 308.873,A -85,B 0,C 180,E1 -14667.589,E2 -14667.589} C_VEL
LIN {X 0,Y 334.06,Z 308.869,A -85,B 0,C 180,E1 -14671.206,E2 -14671.206} C_VEL
LIN {X 0,Y 333.781,Z 308.905,A -85,B 0,C 180,E1 -14673.622,E2 -14673.622} C_VEL
LIN {X 0,Y 333.99,Z 308.881,A -85,B 0,C 180,E1 -14676.04,E2 -14676.04} C_VEL
LIN {X 0,Y 333.917,Z 308.893,A -85,B 0,C 180,E1 -14678.473,E2 -14678.473} C_VEL
LIN {X 0,Y 333.775,Z 308.908,A -85,B 0,C 180,E1 -14682.156,E2 -14682.156} C_VEL
LIN {X 0,Y 333.739,Z 308.915,A -85,B 0,C 180,E1 -14684.638,E2 -14684.638} C_VEL
LIN {X 0,Y 333.699,Z 308.92,A -85,B 0,C 180,E1 -14688.603,E2 -14688.603} C_VEL
LIN {X 0,Y 333.747,Z 309.121,A -85,B 0,C 180,E1 -14691.85,E2 -14691.85} C_VEL
LIN {X 0,Y 335.074,Z 315.825,A -85,B 0,C 180,E1 -14693.855,E2 -14693.855} C_VEL
LIN {X 0,Y 340.387,Z 331.809,A -85,B 0,C 180,E1 -14694.575,E2 -14694.575} C_VEL
LIN {X 0,Y 342.553,Z 343.797,A -85,B 0,C 180,E1 -14694.996,E2 -14694.996} C_VEL
LIN {X 0,Y 340.578,Z 423.664,A -85,B 0,C 180,E1 -14696.855,E2 -14696.855} C_VEL
LIN {X 0,Y 339.891,Z 437.621,A -85,B 0,C 180,E1 -14697.433,E2 -14697.433} C_VEL
LIN {X 0,Y 339.185,Z 450.311,A -85,B 0,C 180,E1 -14698.219,E2 -14698.219} C_VEL
LIN {X 0,Y 338.204,Z 462.36,A -85,B 0,C 180,E1 -14699.216,E2 -14699.216} C_VEL
LIN {X 0,Y 337.221,Z 473.174,A -85,B 0,C 180,E1 -14700.358,E2 -14700.358} C_VEL
LIN {X 0,Y 336.265,Z 483.205,A -85,B 0,C 180,E1 -14701.677,E2 -14701.677} C_VEL
LIN {X 0,Y 335.362,Z 491.706,A -85,B 0,C 180,E1 -14703.042,E2 -14703.042} C_VEL
LIN {X 0,Y 334.46,Z 499.55,A -85,B 0,C 180,E1 -14704.566,E2 -14704.566} C_VEL
LIN {X 0,Y 333.561,Z 507.419,A -85,B 0,C 180,E1 -14706.455,E2 -14706.455} C_VEL
LIN {X 0,Y 332.954,Z 513.163,A -85,B 0,C 180,E1 -14708.179,E2 -14708.179} C_VEL
LIN {X 0,Y 332.6,Z 517.69,A -85,B 0,C 180,E1 -14709.883,E2 -14709.883} C_VEL
LIN {X 0,Y 332.281,Z 521.212,A -85,B 0,C 180,E1 -14711.58,E2 -14711.58} C_VEL
LIN {X 0,Y 332.112,Z 522.516,A -85,B 0,C 180,E1 -14712.351,E2 -14712.351} C_VEL
LIN {X 0,Y 331.287,Z 523.946,A -85,B 0,C 180,E1 -14713.333,E2 -14713.333} C_VEL
LIN {X 0,Y 328.268,Z 525.726,A -85,B 0,C 180,E1 -14714.946,E2 -14714.946} C_VEL
LIN {X 0,Y 325.805,Z 526.612,A -85,B 0,C 180,E1 -14716.266,E2 -14716.266} C_VEL
LIN {X 0,Y 324.773,Z 526.976,A -85,B 0,C 180,E1 -14717.294,E2 -14717.294} C_VEL
LIN {X 0,Y 324.699,Z 527.024,A -85,B 0,C 180,E1 -14717.643,E2 -14717.643} C_VEL
LIN {X 0,Y 324.79,Z 526.719,A -85,B 0,C 180,E1 -14719.521,E2 -14719.521} C_VEL
LIN {X 0,Y 324.992,Z 525.689,A -85,B 0,C 180,E1 -14721.161,E2 -14721.161} C_VEL
LIN {X 0,Y 325.387,Z 523.604,A -85,B 0,C 180,E1 -14723.051,E2 -14723.051} C_VEL
LIN {X 0,Y 325.929,Z 520.341,A -85,B 0,C 180,E1 -14725.025,E2 -14725.025} C_VEL
LIN {X 0,Y 326.692,Z 515.773,A -85,B 0,C 180,E1 -14727.035,E2 -14727.035} C_VEL
LIN {X 0,Y 327.699,Z 509.695,A -85,B 0,C 180,E1 -14729.078,E2 -14729.078} C_VEL
LIN {X 0,Y 328.866,Z 502.837,A -85,B 0,C 180,E1 -14730.885,E2 -14730.885} C_VEL
LIN {X 0,Y 330.274,Z 494.324,A -85,B 0,C 180,E1 -14732.677,E2 -14732.677} C_VEL
LIN {X 0,Y 331.675,Z 485.092,A -85,B 0,C 180,E1 -14734.253,E2 -14734.253} C_VEL
LIN {X 0,Y 333.055,Z 475.677,A -85,B 0,C 180,E1 -14735.556,E2 -14735.556} C_VEL
LIN {X 0,Y 334.498,Z 464.211,A -85,B 0,C 180,E1 -14736.822,E2 -14736.822} C_VEL
LIN {X 0,Y 335.878,Z 451.879,A -85,B 0,C 180,E1 -14737.874,E2 -14737.874} C_VEL
LIN {X 0,Y 336.865,Z 439.166,A -85,B 0,C 180,E1 -14738.686,E2 -14738.686} C_VEL
LIN {X 0,Y 337.614,Z 426.649,A -85,B 0,C 180,E1 -14739.235,E2 -14739.235} C_VEL
LIN {X 0,Y 338.47,Z 400.827,A -85,B 0,C 180,E1 -14739.905,E2 -14739.905} C_VEL
LIN {X 0,Y 340.331,Z 345.463,A -85,B 0,C 180,E1 -14741.244,E2 -14741.244} C_VEL
LIN {X 0,Y 339.056,Z 339.658,A -85,B 0,C 180,E1 -14741.531,E2 -14741.531} C_VEL
LIN {X 0,Y 333.128,Z 325.901,A -85,B 0,C 180,E1 -14742.524,E2 -14742.524} C_VEL
LIN {X 0,Y 328.486,Z 316.323,A -85,B 0,C 180,E1 -14743.347,E2 -14743.347} C_VEL
LIN {X 0,Y 326.767,Z 309.787,A -85,B 0,C 180,E1 -14745.34,E2 -14745.34} C_VEL
LIN {X 0,Y 326.772,Z 309.782,A -85,B 0,C 180,E1 -14748.839,E2 -14748.839} C_VEL
LIN {X 0,Y 326.981,Z 309.756,A -85,B 0,C 180,E1 -14752.59,E2 -14752.59} C_VEL
LIN {X 0,Y 326.778,Z 309.782,A -85,B 0,C 180,E1 -14755.065,E2 -14755.065} C_VEL
LIN {X 0,Y 327.048,Z 309.748,A -85,B 0,C 180,E1 -14757.536,E2 -14757.536} C_VEL
LIN {X 0,Y 327.182,Z 309.73,A -85,B 0,C 180,E1 -14760,E2 -14760} C_VEL
LIN {X 0,Y 327.047,Z 309.747,A -85,B 0,C 180,E1 -14762.463,E2 -14762.463} C_VEL
LIN {X 0,Y 326.957,Z 309.754,A -85,B 0,C 180,E1 -14766.17,E2 -14766.17} C_VEL
LIN {X 0,Y 326.807,Z 309.771,A -85,B 0,C 180,E1 -14769.906,E2 -14769.906} C_VEL
LIN {X 0,Y 326.761,Z 309.774,A -85,B 0,C 180,E1 -14773.685,E2 -14773.685} C_VEL
LIN {X 0,Y 326.665,Z 309.786,A -85,B 0,C 180,E1 -14777.53,E2 -14777.53} C_VEL
LIN {X 0,Y 326.632,Z 309.795,A -85,B 0,C 180,E1 -14780.137,E2 -14780.137} C_VEL
LIN {X 0,Y 326.651,Z 309.789,A -85,B 0,C 180,E1 -14784.129,E2 -14784.129} C_VEL
LIN {X 0,Y 326.685,Z 309.788,A -85,B 0,C 180,E1 -14786.857,E2 -14786.857} C_VEL
LIN {X 0,Y 326.636,Z 309.795,A -85,B 0,C 180,E1 -14790.609,E2 -14790.609} C_VEL
LIN {X 0,Y 326.609,Z 309.798,A -85,B 0,C 180,E1 -14794.019,E2 -14794.019} C_VEL
LIN {X 0,Y 326.629,Z 309.796,A -85,B 0,C 180,E1 -14797.238,E2 -14797.238} C_VEL
LIN {X 0,Y 326.579,Z 309.802,A -85,B 0,C 180,E1 -14801.131,E2 -14801.131} C_VEL
LIN {X 0,Y 326.529,Z 309.813,A -85,B 0,C 180,E1 -14804.742,E2 -14804.742} C_VEL
LIN {X 0,Y 326.578,Z 309.803,A -85,B 0,C 180,E1 -14808.154,E2 -14808.154} C_VEL
LIN {X 0,Y 326.599,Z 309.805,A -85,B 0,C 180,E1 -14811.387,E2 -14811.387} C_VEL
LIN {X 0,Y 326.621,Z 309.806,A -85,B 0,C 180,E1 -14814.851,E2 -14814.851} C_VEL
LIN {X 0,Y 326.629,Z 310.009,A -85,B 0,C 180,E1 -14816.507,E2 -14816.507} C_VEL
LIN {X 0,Y 329.243,Z 319.904,A -85,B 0,C 180,E1 -14819.537,E2 -14819.537} C_VEL
LIN {X 0,Y 331.303,Z 329.159,A -85,B 0,C 180,E1 -14822.18,E2 -14822.18} C_VEL
LIN {X 0,Y 332.156,Z 334.481,A -85,B 0,C 180,E1 -14823.619,E2 -14823.619} C_VEL
LIN {X 0,Y 331.967,Z 336.604,A -85,B 0,C 180,E1 -14824.13,E2 -14824.13} C_VEL
LIN {X 0,Y 336.588,Z 358.706,A -85,B 0,C 180,E1 -14825.228,E2 -14825.228} C_VEL
LIN {X 0,Y 339.218,Z 376.786,A -85,B 0,C 180,E1 -14825.98,E2 -14825.98} C_VEL
LIN {X 0,Y 339.399,Z 381.795,A -85,B 0,C 180,E1 -14826.132,E2 -14826.132} C_VEL
LIN {X 0,Y 337.244,Z 446.938,A -85,B 0,C 180,E1 -14827.726,E2 -14827.726} C_VEL
LIN {X 0,Y 336.29,Z 460.791,A -85,B 0,C 180,E1 -14828.306,E2 -14828.306} C_VEL
LIN {X 0,Y 335.163,Z 472.788,A -85,B 0,C 180,E1 -14829.035,E2 -14829.035} C_VEL
LIN {X 0,Y 333.658,Z 484.527,A -85,B 0,C 180,E1 -14829.983,E2 -14829.983} C_VEL
LIN {X 0,Y 332.211,Z 495.896,A -85,B 0,C 180,E1 -14831.178,E2 -14831.178} C_VEL
LIN {X 0,Y 330.711,Z 506.23,A -85,B 0,C 180,E1 -14832.531,E2 -14832.531} C_VEL
LIN {X 0,Y 329.149,Z 516.404,A -85,B 0,C 180,E1 -14834.202,E2 -14834.202} C_VEL
LIN {X 0,Y 327.786,Z 525.391,A -85,B 0,C 180,E1 -14836.041,E2 -14836.041} C_VEL
LIN {X 0,Y 326.594,Z 532.624,A -85,B 0,C 180,E1 -14837.888,E2 -14837.888} C_VEL
LIN {X 0,Y 325.747,Z 539.246,A -85,B 0,C 180,E1 -14840.06,E2 -14840.06} C_VEL
LIN {X 0,Y 325.263,Z 543.638,A -85,B 0,C 180,E1 -14841.926,E2 -14841.926} C_VEL
LIN {X 0,Y 324.922,Z 547.639,A -85,B 0,C 180,E1 -14844.251,E2 -14844.251} C_VEL
LIN {X 0,Y 324.901,Z 549.856,A -85,B 0,C 180,E1 -14846.279,E2 -14846.279} C_VEL
LIN {X 0,Y 324.858,Z 550.644,A -85,B 0,C 180,E1 -14847.519,E2 -14847.519} C_VEL
LIN {X 0,Y 324.879,Z 551.036,A -85,B 0,C 180,E1 -14848.76,E2 -14848.76} C_VEL
LIN {X 0,Y 324.949,Z 551.031,A -85,B 0,C 180,E1 -14849.999,E2 -14849.999} C_VEL
LIN {X 0,Y 324.895,Z 550.601,A -85,B 0,C 180,E1 -14851.239,E2 -14851.239} C_VEL
LIN {X 0,Y 324.862,Z 549.721,A -85,B 0,C 180,E1 -14852.479,E2 -14852.479} C_VEL
LIN {X 0,Y 324.928,Z 548.434,A -85,B 0,C 180,E1 -14853.72,E2 -14853.72} C_VEL
LIN {X 0,Y 324.927,Z 545.359,A -85,B 0,C 180,E1 -14855.758,E2 -14855.758} C_VEL
LIN {X 0,Y 325.142,Z 541.822,A -85,B 0,C 180,E1 -14857.451,E2 -14857.451} C_VEL
LIN {X 0,Y 325.484,Z 536.812,A -85,B 0,C 180,E1 -14859.319,E2 -14859.319} C_VEL
LIN {X 0,Y 325.978,Z 530.477,A -85,B 0,C 180,E1 -14861.188,E2 -14861.188} C_VEL
LIN {X 0,Y 326.922,Z 522.547,A -85,B 0,C 180,E1 -14863.045,E2 -14863.045} C_VEL
LIN {X 0,Y 327.842,Z 514.422,A -85,B 0,C 180,E1 -14864.588,E2 -14864.588} C_VEL
LIN {X 0,Y 328.875,Z 504.496,A -85,B 0,C 180,E1 -14866.129,E2 -14866.129} C_VEL
LIN {X 0,Y 329.808,Z 494.765,A -85,B 0,C 180,E1 -14867.356,E2 -14867.356} C_VEL
LIN {X 0,Y 330.894,Z 484.338,A -85,B 0,C 180,E1 -14868.416,E2 -14868.416} C_VEL
LIN {X 0,Y 332.061,Z 471.888,A -85,B 0,C 180,E1 -14869.391,E2 -14869.391} C_VEL
LIN {X 0,Y 332.988,Z 458.92,A -85,B 0,C 180,E1 -14870.138,E2 -14870.138} C_VEL
LIN {X 0,Y 333.666,Z 446.425,A -85,B 0,C 180,E1 -14870.618,E2 -14870.618} C_VEL
LIN {X 0,Y 335.17,Z 376.663,A -85,B 0,C 180,E1 -14872.282,E2 -14872.282} C_VEL
LIN {X 0,Y 329.795,Z 339.134,A -85,B 0,C 180,E1 -14873.565,E2 -14873.565} C_VEL
LIN {X 0,Y 330.71,Z 330.125,A -85,B 0,C 180,E1 -14875.826,E2 -14875.826} C_VEL
LIN {X 0,Y 328.706,Z 319.419,A -85,B 0,C 180,E1 -14878.763,E2 -14878.763} C_VEL
LIN {X 0,Y 326.621,Z 309.798,A -85,B 0,C 180,E1 -14881.542,E2 -14881.542} C_VEL
LIN {X 0,Y 326.609,Z 309.798,A -85,B 0,C 180,E1 -14885.519,E2 -14885.519} C_VEL
LIN {X 0,Y 326.608,Z 309.798,A -85,B 0,C 180,E1 -14889.226,E2 -14889.226} C_VEL
LIN {X 0,Y 326.573,Z 309.803,A -85,B 0,C 180,E1 -14892.971,E2 -14892.971} C_VEL
LIN {X 0,Y 326.572,Z 309.804,A -85,B 0,C 180,E1 -14897.027,E2 -14897.027} C_VEL
LIN {X 0,Y 326.608,Z 309.803,A -85,B 0,C 180,E1 -14900.772,E2 -14900.772} C_VEL
LIN {X 0,Y 326.609,Z 309.801,A -85,B 0,C 180,E1 -14904.48,E2 -14904.48} C_VEL
LIN {X 0,Y 326.603,Z 309.799,A -85,B 0,C 180,E1 -14907.455,E2 -14907.455} C_VEL
LIN {X 0,Y 326.642,Z 309.794,A -85,B 0,C 180,E1 -14910.339,E2 -14910.339} C_VEL
LIN {X 0,Y 326.685,Z 309.79,A -85,B 0,C 180,E1 -14914.516,E2 -14914.516} C_VEL
LIN {X 0,Y 326.641,Z 309.794,A -85,B 0,C 180,E1 -14918.545,E2 -14918.545} C_VEL
LIN {X 0,Y 326.739,Z 309.787,A -85,B 0,C 180,E1 -14921.177,E2 -14921.177} C_VEL
LIN {X 0,Y 326.757,Z 309.784,A -85,B 0,C 180,E1 -14925.433,E2 -14925.433} C_VEL
LIN {X 0,Y 326.764,Z 309.779,A -85,B 0,C 180,E1 -14928.839,E2 -14928.839} C_VEL
LIN {X 0,Y 326.974,Z 309.752,A -85,B 0,C 180,E1 -14932.59,E2 -14932.59} C_VEL
LIN {X 0,Y 326.772,Z 309.779,A -85,B 0,C 180,E1 -14935.065,E2 -14935.065} C_VEL
LIN {X 0,Y 327.04,Z 309.749,A -85,B 0,C 180,E1 -14937.537,E2 -14937.537} C_VEL
LIN {X 0,Y 327.191,Z 309.728,A -85,B 0,C 180,E1 -14940,E2 -14940} C_VEL
LIN {X 0,Y 327.041,Z 309.744,A -85,B 0,C 180,E1 -14942.464,E2 -14942.464} C_VEL
LIN {X 0,Y 326.927,Z 309.759,A -85,B 0,C 180,E1 -14946.485,E2 -14946.485} C_VEL
LIN {X 0,Y 326.799,Z 309.779,A -85,B 0,C 180,E1 -14949.907,E2 -14949.907} C_VEL
LIN {X 0,Y 326.754,Z 309.781,A -85,B 0,C 180,E1 -14953.686,E2 -14953.686} C_VEL
LIN {X 0,Y 326.694,Z 309.787,A -85,B 0,C 180,E1 -14957.529,E2 -14957.529} C_VEL
LIN {X 0,Y 326.654,Z 309.797,A -85,B 0,C 180,E1 -14960.136,E2 -14960.136} C_VEL
LIN {X 0,Y 326.629,Z 309.798,A -85,B 0,C 180,E1 -14964.131,E2 -14964.131} C_VEL
LIN {X 0,Y 326.617,Z 309.8,A -85,B 0,C 180,E1 -14968.255,E2 -14968.255} C_VEL
LIN {X 0,Y 326.569,Z 309.804,A -85,B 0,C 180,E1 -14971.098,E2 -14971.098} C_VEL
LIN {X 0,Y 326.604,Z 309.799,A -85,B 0,C 180,E1 -14974.02,E2 -14974.02} C_VEL
LIN {X 0,Y 326.621,Z 309.797,A -85,B 0,C 180,E1 -14977.239,E2 -14977.239} C_VEL
LIN {X 0,Y 326.573,Z 309.805,A -85,B 0,C 180,E1 -14981.132,E2 -14981.132} C_VEL
LIN {X 0,Y 326.525,Z 309.812,A -85,B 0,C 180,E1 -14984.744,E2 -14984.744} C_VEL
LIN {X 0,Y 326.561,Z 309.804,A -85,B 0,C 180,E1 -14988.153,E2 -14988.153} C_VEL
LIN {X 0,Y 326.581,Z 309.804,A -85,B 0,C 180,E1 -14991.387,E2 -14991.387} C_VEL
LIN {X 0,Y 326.619,Z 309.799,A -85,B 0,C 180,E1 -14994.853,E2 -14994.853} C_VEL
LIN {X 0,Y 326.608,Z 309.802,A -85,B 0,C 180,E1 -14997.457,E2 -14997.457} C_VEL
LIN {X 0,Y 326.615,Z 309.797,A -85,B 0,C 180,E1 -15000.338,E2 -15000.338} C_VEL
LIN {X 0,Y 326.642,Z 309.793,A -85,B 0,C 180,E1 -15004.646,E2 -15004.646} C_VEL
LIN {X 0,Y 326.616,Z 309.797,A -85,B 0,C 180,E1 -15008.544,E2 -15008.544} C_VEL
LIN {X 0,Y 326.709,Z 309.787,A -85,B 0,C 180,E1 -15011.176,E2 -15011.176} C_VEL
LIN {X 0,Y 326.766,Z 309.781,A -85,B 0,C 180,E1 -15015.434,E2 -15015.434} C_VEL
LIN {X 0,Y 326.758,Z 309.779,A -85,B 0,C 180,E1 -15018.839,E2 -15018.839} C_VEL
LIN {X 0,Y 326.916,Z 309.76,A -85,B 0,C 180,E1 -15022.59,E2 -15022.59} C_VEL
LIN {X 0,Y 326.744,Z 309.781,A -85,B 0,C 180,E1 -15025.065,E2 -15025.065} C_VEL
LIN {X 0,Y 326.987,Z 309.752,A -85,B 0,C 180,E1 -15027.537,E2 -15027.537} C_VEL
LIN {X 0,Y 327.029,Z 309.745,A -85,B 0,C 180,E1 -15031.232,E2 -15031.232} C_VEL
LIN {X 0,Y 326.731,Z 309.784,A -85,B 0,C 180,E1 -15033.701,E2 -15033.701} C_VEL
LIN {X 0,Y 326.944,Z 309.76,A -85,B 0,C 180,E1 -15036.171,E2 -15036.171} C_VEL
LIN {X 0,Y 326.78,Z 309.778,A -85,B 0,C 180,E1 -15039.908,E2 -15039.908} C_VEL
LIN {X 0,Y 326.726,Z 309.783,A -85,B 0,C 180,E1 -15043.687,E2 -15043.687} C_VEL
LIN {X 0,Y 326.633,Z 309.795,A -85,B 0,C 180,E1 -15047.532,E2 -15047.532} C_VEL
LIN {X 0,Y 326.667,Z 309.863,A -85,B 0,C 180,E1 -15051.515,E2 -15051.515} C_VEL
LIN {X 0,Y 327.875,Z 315.947,A -85,B 0,C 180,E1 -15053.402,E2 -15053.402} C_VEL
LIN {X 0,Y 333.88,Z 333.801,A -85,B 0,C 180,E1 -15054.235,E2 -15054.235} C_VEL
LIN {X 0,Y 335.83,Z 344.464,A -85,B 0,C 180,E1 -15054.62,E2 -15054.62} C_VEL
LIN {X 0,Y 333.794,Z 424.02,A -85,B 0,C 180,E1 -15056.515,E2 -15056.515} C_VEL
LIN {X 0,Y 333.076,Z 437.973,A -85,B 0,C 180,E1 -15057.106,E2 -15057.106} C_VEL
LIN {X 0,Y 332.36,Z 450.466,A -85,B 0,C 180,E1 -15057.895,E2 -15057.895} C_VEL
LIN {X 0,Y 331.413,Z 461.833,A -85,B 0,C 180,E1 -15058.845,E2 -15058.845} C_VEL
LIN {X 0,Y 330.355,Z 473.143,A -85,B 0,C 180,E1 -15060.051,E2 -15060.051} C_VEL
LIN {X 0,Y 329.345,Z 483.243,A -85,B 0,C 180,E1 -15061.396,E2 -15061.396} C_VEL
LIN {X 0,Y 328.255,Z 493.231,A -85,B 0,C 180,E1 -15063.059,E2 -15063.059} C_VEL
LIN {X 0,Y 327.173,Z 502.175,A -85,B 0,C 180,E1 -15064.906,E2 -15064.906} C_VEL
LIN {X 0,Y 326.347,Z 509.094,A -85,B 0,C 180,E1 -15066.699,E2 -15066.699} C_VEL
LIN {X 0,Y 325.743,Z 515.282,A -85,B 0,C 180,E1 -15068.733,E2 -15068.733} C_VEL
LIN {X 0,Y 325.299,Z 520.247,A -85,B 0,C 180,E1 -15070.872,E2 -15070.872} C_VEL
LIN {X 0,Y 324.956,Z 523.285,A -85,B 0,C 180,E1 -15072.664,E2 -15072.664} C_VEL
LIN {X 0,Y 324.736,Z 525.367,A -85,B 0,C 180,E1 -15074.422,E2 -15074.422} C_VEL
LIN {X 0,Y 324.679,Z 526.604,A -85,B 0,C 180,E1 -15076.157,E2 -15076.157} C_VEL
LIN {X 0,Y 324.699,Z 527.024,A -85,B 0,C 180,E1 -15077.643,E2 -15077.643} C_VEL
LIN {X 0,Y 324.078,Z 527.05,A -85,B 0,C 180,E1 -15078.68,E2 -15078.68} C_VEL
LIN {X 0,Y 321.366,Z 526.527,A -85,B 0,C 180,E1 -15080.371,E2 -15080.371} C_VEL
LIN {X 0,Y 319.15,Z 525.56,A -85,B 0,C 180,E1 -15081.731,E2 -15081.731} C_VEL
LIN {X 0,Y 318.323,Z 524.516,A -85,B 0,C 180,E1 -15082.771,E2 -15082.771} C_VEL
LIN {X 0,Y 318.323,Z 524.059,A -85,B 0,C 180,E1 -15083.119,E2 -15083.119} C_VEL
LIN {X 0,Y 318.865,Z 521.103,A -85,B 0,C 180,E1 -15085.036,E2 -15085.036} C_VEL
LIN {X 0,Y 319.823,Z 515.735,A -85,B 0,C 180,E1 -15087.463,E2 -15087.463} C_VEL
LIN {X 0,Y 320.741,Z 510.472,A -85,B 0,C 180,E1 -15089.274,E2 -15089.274} C_VEL
LIN {X 0,Y 321.78,Z 504.687,A -85,B 0,C 180,E1 -15090.885,E2 -15090.885} C_VEL
LIN {X 0,Y 323.365,Z 495.966,A -85,B 0,C 180,E1 -15092.844,E2 -15092.844} C_VEL
LIN {X 0,Y 324.892,Z 486.292,A -85,B 0,C 180,E1 -15094.567,E2 -15094.567} C_VEL
LIN {X 0,Y 326.516,Z 475.897,A -85,B 0,C 180,E1 -15096.046,E2 -15096.046} C_VEL
LIN {X 0,Y 328,Z 464.625,A -85,B 0,C 180,E1 -15097.313,E2 -15097.313} C_VEL
LIN {X 0,Y 329.37,Z 453.117,A -85,B 0,C 180,E1 -15098.32,E2 -15098.32} C_VEL
LIN {X 0,Y 330.378,Z 441.309,A -85,B 0,C 180,E1 -15099.118,E2 -15099.118} C_VEL
LIN {X 0,Y 331.146,Z 429.021,A -85,B 0,C 180,E1 -15099.709,E2 -15099.709} C_VEL
LIN {X 0,Y 331.907,Z 411.202,A -85,B 0,C 180,E1 -15100.217,E2 -15100.217} C_VEL
LIN {X 0,Y 334.184,Z 346.964,A -85,B 0,C 180,E1 -15101.81,E2 -15101.81} C_VEL
LIN {X 0,Y 333.229,Z 342.526,A -85,B 0,C 180,E1 -15102.034,E2 -15102.034} C_VEL
LIN {X 0,Y 327.288,Z 328.666,A -85,B 0,C 180,E1 -15103.068,E2 -15103.068} C_VEL
LIN {X 0,Y 321.352,Z 316.773,A -85,B 0,C 180,E1 -15104.134,E2 -15104.134} C_VEL
LIN {X 0,Y 319.724,Z 310.664,A -85,B 0,C 180,E1 -15106.088,E2 -15106.088} C_VEL
LIN {X 0,Y 319.76,Z 310.654,A -85,B 0,C 180,E1 -15109.873,E2 -15109.873} C_VEL
LIN {X 0,Y 319.935,Z 310.634,A -85,B 0,C 180,E1 -15112.426,E2 -15112.426} C_VEL
LIN {X 0,Y 319.748,Z 310.658,A -85,B 0,C 180,E1 -15114.956,E2 -15114.956} C_VEL
LIN {X 0,Y 319.991,Z 310.627,A -85,B 0,C 180,E1 -15117.482,E2 -15117.482} C_VEL
LIN {X 0,Y 320.134,Z 310.607,A -85,B 0,C 180,E1 -15120,E2 -15120} C_VEL
LIN {X 0,Y 319.991,Z 310.626,A -85,B 0,C 180,E1 -15122.517,E2 -15122.517} C_VEL
LIN {X 0,Y 319.913,Z 310.63,A -85,B 0,C 180,E1 -15126.306,E2 -15126.306} C_VEL
LIN {X 0,Y 319.754,Z 310.649,A -85,B 0,C 180,E1 -15130.127,E2 -15130.127} C_VEL
LIN {X 0,Y 319.734,Z 310.65,A -85,B 0,C 180,E1 -15133.992,E2 -15133.992} C_VEL
LIN {X 0,Y 319.626,Z 310.664,A -85,B 0,C 180,E1 -15137.929,E2 -15137.929} C_VEL
LIN {X 0,Y 319.569,Z 310.673,A -85,B 0,C 180,E1 -15141.954,E2 -15141.954} C_VEL
LIN {X 0,Y 319.636,Z 310.667,A -85,B 0,C 180,E1 -15146.088,E2 -15146.088} C_VEL
LIN {X 0,Y 319.582,Z 310.671,A -85,B 0,C 180,E1 -15148.934,E2 -15148.934} C_VEL
LIN {X 0,Y 319.532,Z 310.676,A -85,B 0,C 180,E1 -15151.862,E2 -15151.862} C_VEL
LIN {X 0,Y 319.582,Z 310.674,A -85,B 0,C 180,E1 -15155.543,E2 -15155.543} C_VEL
LIN {X 0,Y 319.56,Z 310.679,A -85,B 0,C 180,E1 -15159.668,E2 -15159.668} C_VEL
LIN {X 0,Y 319.523,Z 310.682,A -85,B 0,C 180,E1 -15163.46,E2 -15163.46} C_VEL
LIN {X 0,Y 319.556,Z 310.681,A -85,B 0,C 180,E1 -15167.016,E2 -15167.016} C_VEL
LIN {X 0,Y 319.549,Z 310.68,A -85,B 0,C 180,E1 -15170.371,E2 -15170.371} C_VEL
LIN {X 0,Y 319.582,Z 310.684,A -85,B 0,C 180,E1 -15174.457,E2 -15174.457} C_VEL
LIN {X 0,Y 319.575,Z 310.738,A -85,B 0,C 180,E1 -15175.747,E2 -15175.747} C_VEL
LIN {X 0,Y 322.437,Z 321.591,A -85,B 0,C 180,E1 -15179.188,E2 -15179.188} C_VEL
LIN {X 0,Y 324.684,Z 331.708,A -85,B 0,C 180,E1 -15182.15,E2 -15182.15} C_VEL
LIN {X 0,Y 325.412,Z 336.359,A -85,B 0,C 180,E1 -15183.416,E2 -15183.416} C_VEL
LIN {X 0,Y 329.558,Z 355.341,A -85,B 0,C 180,E1 -15184.424,E2 -15184.424} C_VEL
LIN {X 0,Y 332.783,Z 375.735,A -85,B 0,C 180,E1 -15185.336,E2 -15185.336} C_VEL
LIN {X 0,Y 333.205,Z 381.232,A -85,B 0,C 180,E1 -15185.534,E2 -15185.534} C_VEL
LIN {X 0,Y 330.886,Z 447.095,A -85,B 0,C 180,E1 -15187.192,E2 -15187.192} C_VEL
LIN {X 0,Y 329.886,Z 460.796,A -85,B 0,C 180,E1 -15187.78,E2 -15187.78} C_VEL
LIN {X 0,Y 328.687,Z 472.704,A -85,B 0,C 180,E1 -15188.52,E2 -15188.52} C_VEL
LIN {X 0,Y 327.026,Z 485.18,A -85,B 0,C 180,E1 -15189.56,E2 -15189.56} C_VEL
LIN {X 0,Y 325.527,Z 496.386,A -85,B 0,C 180,E1 -15190.777,E2 -15190.777} C_VEL
LIN {X 0,Y 323.947,Z 506.564,A -85,B 0,C 180,E1 -15192.155,E2 -15192.155} C_VEL
LIN {X 0,Y 322.456,Z 515.833,A -85,B 0,C 180,E1 -15193.714,E2 -15193.714} C_VEL
LIN {X 0,Y 321.141,Z 524.107,A -85,B 0,C 180,E1 -15195.423,E2 -15195.423} C_VEL
LIN {X 0,Y 319.813,Z 531.522,A -85,B 0,C 180,E1 -15197.305,E2 -15197.305} C_VEL
LIN {X 0,Y 318.931,Z 537.505,A -85,B 0,C 180,E1 -15199.204,E2 -15199.204} C_VEL
LIN {X 0,Y 318.357,Z 542.234,A -85,B 0,C 180,E1 -15201.11,E2 -15201.11} C_VEL
LIN {X 0,Y 317.988,Z 545.85,A -85,B 0,C 180,E1 -15203.017,E2 -15203.017} C_VEL
LIN {X 0,Y 317.807,Z 548.444,A -85,B 0,C 180,E1 -15204.924,E2 -15204.924} C_VEL
LIN {X 0,Y 317.808,Z 549.642,A -85,B 0,C 180,E1 -15206.195,E2 -15206.195} C_VEL
LIN {X 0,Y 317.778,Z 550.408,A -85,B 0,C 180,E1 -15207.464,E2 -15207.464} C_VEL
LIN {X 0,Y 317.788,Z 550.778,A -85,B 0,C 180,E1 -15208.732,E2 -15208.732} C_VEL
LIN {X 0,Y 317.854,Z 550.752,A -85,B 0,C 180,E1 -15209.999,E2 -15209.999} C_VEL
LIN {X 0,Y 317.802,Z 550.278,A -85,B 0,C 180,E1 -15211.266,E2 -15211.266} C_VEL
LIN {X 0,Y 317.783,Z 549.377,A -85,B 0,C 180,E1 -15212.534,E2 -15212.534} C_VEL
LIN {X 0,Y 317.833,Z 548.067,A -85,B 0,C 180,E1 -15213.803,E2 -15213.803} C_VEL
LIN {X 0,Y 317.847,Z 545.214,A -85,B 0,C 180,E1 -15215.728,E2 -15215.728} C_VEL
LIN {X 0,Y 318.061,Z 541.356,A -85,B 0,C 180,E1 -15217.618,E2 -15217.618} C_VEL
LIN {X 0,Y 318.422,Z 536.29,A -85,B 0,C 180,E1 -15219.527,E2 -15219.527} C_VEL
LIN {X 0,Y 318.974,Z 529.888,A -85,B 0,C 180,E1 -15221.437,E2 -15221.437} C_VEL
LIN {X 0,Y 319.972,Z 521.852,A -85,B 0,C 180,E1 -15223.333,E2 -15223.333} C_VEL
LIN {X 0,Y 320.931,Z 513.637,A -85,B 0,C 180,E1 -15224.91,E2 -15224.91} C_VEL
LIN {X 0,Y 321.994,Z 503.598,A -85,B 0,C 180,E1 -15226.483,E2 -15226.483} C_VEL
LIN {X 0,Y 323.153,Z 492.304,A -85,B 0,C 180,E1 -15227.889,E2 -15227.889} C_VEL
LIN {X 0,Y 324.304,Z 481.288,A -85,B 0,C 180,E1 -15228.969,E2 -15228.969} C_VEL
LIN {X 0,Y 325.424,Z 469.189,A -85,B 0,C 180,E1 -15229.885,E2 -15229.885} C_VEL
LIN {X 0,Y 326.31,Z 456.774,A -85,B 0,C 180,E1 -15230.568,E2 -15230.568} C_VEL
LIN {X 0,Y 326.974,Z 442.929,A -85,B 0,C 180,E1 -15231.06,E2 -15231.06} C_VEL
LIN {X 0,Y 328.382,Z 377.243,A -85,B 0,C 180,E1 -15232.657,E2 -15232.657} C_VEL
LIN {X 0,Y 322.976,Z 338.857,A -85,B 0,C 180,E1 -15234.004,E2 -15234.004} C_VEL
LIN {X 0,Y 323.748,Z 332.119,A -85,B 0,C 180,E1 -15235.731,E2 -15235.731} C_VEL
LIN {X 0,Y 322.722,Z 325.473,A -85,B 0,C 180,E1 -15237.565,E2 -15237.565} C_VEL
LIN {X 0,Y 320.113,Z 313.196,A -85,B 0,C 180,E1 -15241.104,E2 -15241.104} C_VEL
LIN {X 0,Y 319.571,Z 310.68,A -85,B 0,C 180,E1 -15241.856,E2 -15241.856} C_VEL
LIN {X 0,Y 319.577,Z 310.675,A -85,B 0,C 180,E1 -15245.542,E2 -15245.542} C_VEL
LIN {X 0,Y 319.57,Z 310.678,A -85,B 0,C 180,E1 -15248.007,E2 -15248.007} C_VEL
LIN {X 0,Y 319.522,Z 310.681,A -85,B 0,C 180,E1 -15251.596,E2 -15251.596} C_VEL
LIN {X 0,Y 319.485,Z 310.685,A -85,B 0,C 180,E1 -15255.257,E2 -15255.257} C_VEL
LIN {X 0,Y 319.525,Z 310.685,A -85,B 0,C 180,E1 -15258.711,E2 -15258.711} C_VEL
LIN {X 0,Y 319.574,Z 310.677,A -85,B 0,C 180,E1 -15262.343,E2 -15262.343} C_VEL
LIN {X 0,Y 319.556,Z 310.679,A -85,B 0,C 180,E1 -15265.123,E2 -15265.123} C_VEL
LIN {X 0,Y 319.561,Z 310.678,A -85,B 0,C 180,E1 -15269.059,E2 -15269.059} C_VEL
LIN {X 0,Y 319.6,Z 310.672,A -85,B 0,C 180,E1 -15272.498,E2 -15272.498} C_VEL
LIN {X 0,Y 319.6,Z 310.674,A -85,B 0,C 180,E1 -15275.304,E2 -15275.304} C_VEL
LIN {X 0,Y 319.592,Z 310.672,A -85,B 0,C 180,E1 -15278.048,E2 -15278.048} C_VEL
LIN {X 0,Y 319.684,Z 310.664,A -85,B 0,C 180,E1 -15280.962,E2 -15280.962} C_VEL
LIN {X 0,Y 319.725,Z 310.661,A -85,B 0,C 180,E1 -15285.276,E2 -15285.276} C_VEL
LIN {X 0,Y 319.752,Z 310.654,A -85,B 0,C 180,E1 -15289.873,E2 -15289.873} C_VEL
LIN {X 0,Y 319.927,Z 310.63,A -85,B 0,C 180,E1 -15292.426,E2 -15292.426} C_VEL
LIN {X 0,Y 319.741,Z 310.654,A -85,B 0,C 180,E1 -15294.956,E2 -15294.956} C_VEL
LIN {X 0,Y 319.984,Z 310.627,A -85,B 0,C 180,E1 -15297.483,E2 -15297.483} C_VEL
LIN {X 0,Y 320.143,Z 310.606,A -85,B 0,C 180,E1 -15300,E2 -15300} C_VEL
LIN {X 0,Y 319.984,Z 310.623,A -85,B 0,C 180,E1 -15302.518,E2 -15302.518} C_VEL
LIN {X 0,Y 319.893,Z 310.635,A -85,B 0,C 180,E1 -15306.469,E2 -15306.469} C_VEL
LIN {X 0,Y 319.747,Z 310.656,A -85,B 0,C 180,E1 -15310.128,E2 -15310.128} C_VEL
LIN {X 0,Y 319.726,Z 310.655,A -85,B 0,C 180,E1 -15314.725,E2 -15314.725} C_VEL
LIN {X 0,Y 319.684,Z 310.66,A -85,B 0,C 180,E1 -15319.038,E2 -15319.038} C_VEL
LIN {X 0,Y 319.548,Z 310.676,A -85,B 0,C 180,E1 -15323.322,E2 -15323.322} C_VEL
LIN {X 0,Y 319.567,Z 310.676,A -85,B 0,C 180,E1 -15326.094,E2 -15326.094} C_VEL
LIN {X 0,Y 319.548,Z 310.679,A -85,B 0,C 180,E1 -15328.938,E2 -15328.938} C_VEL
LIN {X 0,Y 319.52,Z 310.681,A -85,B 0,C 180,E1 -15331.864,E2 -15331.864} C_VEL
LIN {X 0,Y 319.576,Z 310.673,A -85,B 0,C 180,E1 -15335.544,E2 -15335.544} C_VEL
LIN {X 0,Y 319.556,Z 310.675,A -85,B 0,C 180,E1 -15339.67,E2 -15339.67} C_VEL
LIN {X 0,Y 319.519,Z 310.682,A -85,B 0,C 180,E1 -15343.462,E2 -15343.462} C_VEL
LIN {X 0,Y 319.55,Z 310.683,A -85,B 0,C 180,E1 -15347.017,E2 -15347.017} C_VEL
LIN {X 0,Y 319.544,Z 310.678,A -85,B 0,C 180,E1 -15350.372,E2 -15350.372} C_VEL
LIN {X 0,Y 319.579,Z 310.673,A -85,B 0,C 180,E1 -15354.458,E2 -15354.458} C_VEL
LIN {X 0,Y 319.524,Z 310.68,A -85,B 0,C 180,E1 -15358.138,E2 -15358.138} C_VEL
LIN {X 0,Y 319.569,Z 310.678,A -85,B 0,C 180,E1 -15361.606,E2 -15361.606} C_VEL
LIN {X 0,Y 319.574,Z 310.678,A -85,B 0,C 180,E1 -15365.302,E2 -15365.302} C_VEL
LIN {X 0,Y 319.567,Z 310.676,A -85,B 0,C 180,E1 -15368.047,E2 -15368.047} C_VEL
LIN {X 0,Y 319.627,Z 310.67,A -85,B 0,C 180,E1 -15372.072,E2 -15372.072} C_VEL
LIN {X 0,Y 319.735,Z 310.658,A -85,B 0,C 180,E1 -15376.009,E2 -15376.009} C_VEL
LIN {X 0,Y 319.737,Z 310.66,A -85,B 0,C 180,E1 -15379.873,E2 -15379.873} C_VEL
LIN {X 0,Y 319.901,Z 310.636,A -85,B 0,C 180,E1 -15383.694,E2 -15383.694} C_VEL
LIN {X 0,Y 319.998,Z 310.622,A -85,B 0,C 180,E1 -15388.742,E2 -15388.742} C_VEL
LIN {X 0,Y 319.934,Z 310.633,A -85,B 0,C 180,E1 -15392.519,E2 -15392.519} C_VEL
LIN {X 0,Y 319.902,Z 310.639,A -85,B 0,C 180,E1 -15396.307,E2 -15396.307} C_VEL
LIN {X 0,Y 319.732,Z 310.657,A -85,B 0,C 180,E1 -15400.129,E2 -15400.129} C_VEL
LIN {X 0,Y 319.697,Z 310.66,A -85,B 0,C 180,E1 -15403.994,E2 -15403.994} C_VEL
LIN {X 0,Y 319.589,Z 310.673,A -85,B 0,C 180,E1 -15407.932,E2 -15407.932} C_VEL
LIN {X 0,Y 319.585,Z 310.677,A -85,B 0,C 180,E1 -15411.192,E2 -15411.192} C_VEL
LIN {X 0,Y 320.703,Z 316.185,A -85,B 0,C 180,E1 -15412.941,E2 -15412.941} C_VEL
LIN {X 0,Y 327.262,Z 335.259,A -85,B 0,C 180,E1 -15413.871,E2 -15413.871} C_VEL
LIN {X 0,Y 329.116,Z 345.527,A -85,B 0,C 180,E1 -15414.249,E2 -15414.249} C_VEL
LIN {X 0,Y 327.004,Z 423.598,A -85,B 0,C 180,E1 -15416.145,E2 -15416.145} C_VEL
LIN {X 0,Y 326.292,Z 437.581,A -85,B 0,C 180,E1 -15416.74,E2 -15416.74} C_VEL
LIN {X 0,Y 325.605,Z 449.752,A -85,B 0,C 180,E1 -15417.506,E2 -15417.506} C_VEL
LIN {X 0,Y 324.534,Z 462.019,A -85,B 0,C 180,E1 -15418.541,E2 -15418.541} C_VEL
LIN {X 0,Y 323.434,Z 473.489,A -85,B 0,C 180,E1 -15419.789,E2 -15419.789} C_VEL
LIN {X 0,Y 322.383,Z 483.701,A -85,B 0,C 180,E1 -15421.182,E2 -15421.182} C_VEL
LIN {X 0,Y 321.313,Z 493.111,A -85,B 0,C 180,E1 -15422.776,E2 -15422.776} C_VEL
LIN {X 0,Y 320.271,Z 501.376,A -85,B 0,C 180,E1 -15424.492,E2 -15424.492} C_VEL
LIN {X 0,Y 319.363,Z 508.985,A -85,B 0,C 180,E1 -15426.454,E2 -15426.454} C_VEL
LIN {X 0,Y 318.791,Z 514.149,A -85,B 0,C 180,E1 -15428.119,E2 -15428.119} C_VEL
LIN {X 0,Y 318.43,Z 518.351,A -85,B 0,C 180,E1 -15429.796,E2 -15429.796} C_VEL
LIN {X 0,Y 318.109,Z 521.749,A -85,B 0,C 180,E1 -15431.514,E2 -15431.514} C_VEL
LIN {X 0,Y 317.774,Z 524.374,A -85,B 0,C 180,E1 -15433.284,E2 -15433.284} C_VEL
LIN {X 0,Y 317.616,Z 526.177,A -85,B 0,C 180,E1 -15435.079,E2 -15435.079} C_VEL
LIN {X 0,Y 317.585,Z 527.156,A -85,B 0,C 180,E1 -15436.91,E2 -15436.91} C_VEL
LIN {X 0,Y 317.649,Z 527.256,A -85,B 0,C 180,E1 -15438.786,E2 -15438.786} C_VEL
LIN {X 0,Y 317.834,Z 526.44,A -85,B 0,C 180,E1 -15440.708,E2 -15440.708} C_VEL
LIN {X 0,Y 318.222,Z 524.643,A -85,B 0,C 180,E1 -15442.662,E2 -15442.662} C_VEL
LIN {X 0,Y 318.323,Z 524.059,A -85,B 0,C 180,E1 -15443.119,E2 -15443.119} C_VEL
LIN {X 0,Y 317.927,Z 522.674,A -85,B 0,C 180,E1 -15444.151,E2 -15444.151} C_VEL
LIN {X 0,Y 315.595,Z 520.011,A -85,B 0,C 180,E1 -15445.828,E2 -15445.828} C_VEL
LIN {X 0,Y 313.406,Z 516.703,A -85,B 0,C 180,E1 -15447.488,E2 -15447.488} C_VEL
LIN {X 0,Y 313.24,Z 514.23,A -85,B 0,C 180,E1 -15448.473,E2 -15448.473} C_VEL
LIN {X 0,Y 314.535,Z 507.461,A -85,B 0,C 180,E1 -15450.625,E2 -15450.625} C_VEL
LIN {X 0,Y 316.034,Z 499.913,A -85,B 0,C 180,E1 -15452.504,E2 -15452.504} C_VEL
LIN {X 0,Y 317.656,Z 490.572,A -85,B 0,C 180,E1 -15454.362,E2 -15454.362} C_VEL
LIN {X 0,Y 319.317,Z 480.457,A -85,B 0,C 180,E1 -15455.972,E2 -15455.972} C_VEL
LIN {X 0,Y 320.944,Z 469.655,A -85,B 0,C 180,E1 -15457.334,E2 -15457.334} C_VEL
LIN {X 0,Y 322.436,Z 457.977,A -85,B 0,C 180,E1 -15458.499,E2 -15458.499} C_VEL
LIN {X 0,Y 323.724,Z 445.906,A -85,B 0,C 180,E1 -15459.419,E2 -15459.419} C_VEL
LIN {X 0,Y 324.664,Z 432.662,A -85,B 0,C 180,E1 -15460.148,E2 -15460.148} C_VEL
LIN {X 0,Y 325.358,Z 419.688,A -85,B 0,C 180,E1 -15460.602,E2 -15460.602} C_VEL
LIN {X 0,Y 328.019,Z 347.853,A -85,B 0,C 180,E1 -15462.418,E2 -15462.418} C_VEL
LIN {X 0,Y 326.926,Z 344.037,A -85,B 0,C 180,E1 -15462.646,E2 -15462.646} C_VEL
LIN {X 0,Y 320.988,Z 330.435,A -85,B 0,C 180,E1 -15463.732,E2 -15463.732} C_VEL
LIN {X 0,Y 314.235,Z 317.121,A -85,B 0,C 180,E1 -15465.013,E2 -15465.013} C_VEL
LIN {X 0,Y 312.664,Z 311.541,A -85,B 0,C 180,E1 -15466.886,E2 -15466.886} C_VEL
LIN {X 0,Y 312.837,Z 311.517,A -85,B 0,C 180,E1 -15471.296,E2 -15471.296} C_VEL
LIN {X 0,Y 312.912,Z 311.507,A -85,B 0,C 180,E1 -15473.552,E2 -15473.552} C_VEL
LIN {X 0,Y 312.938,Z 311.506,A -85,B 0,C 180,E1 -15477.425,E2 -15477.425} C_VEL
LIN {X 0,Y 313.087,Z 311.485,A -85,B 0,C 180,E1 -15480,E2 -15480} C_VEL
LIN {X 0,Y 312.937,Z 311.504,A -85,B 0,C 180,E1 -15482.574,E2 -15482.574} C_VEL
LIN {X 0,Y 312.856,Z 311.508,A -85,B 0,C 180,E1 -15486.449,E2 -15486.449} C_VEL
LIN {X 0,Y 312.758,Z 311.524,A -85,B 0,C 180,E1 -15489.05,E2 -15489.05} C_VEL
LIN {X 0,Y 312.636,Z 311.535,A -85,B 0,C 180,E1 -15492.991,E2 -15492.991} C_VEL
LIN {X 0,Y 312.627,Z 311.542,A -85,B 0,C 180,E1 -15495.65,E2 -15495.65} C_VEL
LIN {X 0,Y 312.561,Z 311.55,A -85,B 0,C 180,E1 -15499.711,E2 -15499.711} C_VEL
LIN {X 0,Y 312.528,Z 311.555,A -85,B 0,C 180,E1 -15502.78,E2 -15502.78} C_VEL
LIN {X 0,Y 312.604,Z 311.543,A -85,B 0,C 180,E1 -15505.935,E2 -15505.935} C_VEL
LIN {X 0,Y 312.54,Z 311.552,A -85,B 0,C 180,E1 -15509.65,E2 -15509.65} C_VEL
LIN {X 0,Y 312.521,Z 311.554,A -85,B 0,C 180,E1 -15513.688,E2 -15513.688} C_VEL
LIN {X 0,Y 312.522,Z 311.551,A -85,B 0,C 180,E1 -15517.386,E2 -15517.386} C_VEL
LIN {X 0,Y 312.492,Z 311.556,A -85,B 0,C 180,E1 -15520.709,E2 -15520.709} C_VEL
LIN {X 0,Y 312.453,Z 311.566,A -85,B 0,C 180,E1 -15524.209,E2 -15524.209} C_VEL
LIN {X 0,Y 312.486,Z 311.558,A -85,B 0,C 180,E1 -15527.918,E2 -15527.918} C_VEL
LIN {X 0,Y 312.5,Z 311.561,A -85,B 0,C 180,E1 -15530.971,E2 -15530.971} C_VEL
LIN {X 0,Y 312.56,Z 311.745,A -85,B 0,C 180,E1 -15535.013,E2 -15535.013} C_VEL
LIN {X 0,Y 315.463,Z 322.577,A -85,B 0,C 180,E1 -15538.587,E2 -15538.587} C_VEL
LIN {X 0,Y 317.719,Z 332.471,A -85,B 0,C 180,E1 -15541.603,E2 -15541.603} C_VEL
LIN {X 0,Y 318.307,Z 335.833,A -85,B 0,C 180,E1 -15542.57,E2 -15542.57} C_VEL
LIN {X 0,Y 320.254,Z 341.433,A -85,B 0,C 180,E1 -15542.984,E2 -15542.984} C_VEL
LIN {X 0,Y 324.338,Z 361.447,A -85,B 0,C 180,E1 -15544.057,E2 -15544.057} C_VEL
LIN {X 0,Y 326.977,Z 380.107,A -85,B 0,C 180,E1 -15544.88,E2 -15544.88} C_VEL
LIN {X 0,Y 324.91,Z 441.649,A -85,B 0,C 180,E1 -15546.453,E2 -15546.453} C_VEL
LIN {X 0,Y 323.992,Z 455.863,A -85,B 0,C 180,E1 -15546.974,E2 -15546.974} C_VEL
LIN {X 0,Y 322.729,Z 468.378,A -85,B 0,C 180,E1 -15547.682,E2 -15547.682} C_VEL
LIN {X 0,Y 321.173,Z 481.009,A -85,B 0,C 180,E1 -15548.666,E2 -15548.666} C_VEL
LIN {X 0,Y 319.709,Z 491.654,A -85,B 0,C 180,E1 -15549.743,E2 -15549.743} C_VEL
LIN {X 0,Y 317.893,Z 502.66,A -85,B 0,C 180,E1 -15551.135,E2 -15551.135} C_VEL
LIN {X 0,Y 316.398,Z 511.656,A -85,B 0,C 180,E1 -15552.55,E2 -15552.55} C_VEL
LIN {X 0,Y 314.98,Z 520.15,A -85,B 0,C 180,E1 -15554.181,E2 -15554.181} C_VEL
LIN {X 0,Y 313.575,Z 528.119,A -85,B 0,C 180,E1 -15556.058,E2 -15556.058} C_VEL
LIN {X 0,Y 312.514,Z 533.681,A -85,B 0,C 180,E1 -15557.663,E2 -15557.663} C_VEL
LIN {X 0,Y 311.694,Z 539.148,A -85,B 0,C 180,E1 -15559.607,E2 -15559.607} C_VEL
LIN {X 0,Y 311.152,Z 543.432,A -85,B 0,C 180,E1 -15561.557,E2 -15561.557} C_VEL
LIN {X 0,Y 310.823,Z 546.652,A -85,B 0,C 180,E1 -15563.508,E2 -15563.508} C_VEL
LIN {X 0,Y 310.71,Z 548.27,A -85,B 0,C 180,E1 -15564.808,E2 -15564.808} C_VEL
LIN {X 0,Y 310.719,Z 549.427,A -85,B 0,C 180,E1 -15566.108,E2 -15566.108} C_VEL
LIN {X 0,Y 310.7,Z 550.172,A -85,B 0,C 180,E1 -15567.406,E2 -15567.406} C_VEL
LIN {X 0,Y 310.699,Z 550.521,A -85,B 0,C 180,E1 -15568.703,E2 -15568.703} C_VEL
LIN {X 0,Y 310.76,Z 550.465,A -85,B 0,C 180,E1 -15569.999,E2 -15569.999} C_VEL
LIN {X 0,Y 310.713,Z 549.95,A -85,B 0,C 180,E1 -15571.295,E2 -15571.295} C_VEL
LIN {X 0,Y 310.706,Z 549.025,A -85,B 0,C 180,E1 -15572.592,E2 -15572.592} C_VEL
LIN {X 0,Y 310.742,Z 547.69,A -85,B 0,C 180,E1 -15573.89,E2 -15573.89} C_VEL
LIN {X 0,Y 310.765,Z 545.061,A -85,B 0,C 180,E1 -15575.693,E2 -15575.693} C_VEL
LIN {X 0,Y 311.002,Z 540.868,A -85,B 0,C 180,E1 -15577.792,E2 -15577.792} C_VEL
LIN {X 0,Y 311.475,Z 534.745,A -85,B 0,C 180,E1 -15580.07,E2 -15580.07} C_VEL
LIN {X 0,Y 312.126,Z 527.987,A -85,B 0,C 180,E1 -15582.021,E2 -15582.021} C_VEL
LIN {X 0,Y 313.137,Z 519.586,A -85,B 0,C 180,E1 -15583.961,E2 -15583.961} C_VEL
LIN {X 0,Y 314.188,Z 510.948,A -85,B 0,C 180,E1 -15585.57,E2 -15585.57} C_VEL
LIN {X 0,Y 315.343,Z 500.25,A -85,B 0,C 180,E1 -15587.175,E2 -15587.175} C_VEL
LIN {X 0,Y 316.505,Z 489.679,A -85,B 0,C 180,E1 -15588.446,E2 -15588.446} C_VEL
LIN {X 0,Y 317.752,Z 478.059,A -85,B 0,C 180,E1 -15589.543,E2 -15589.543} C_VEL
LIN {X 0,Y 318.901,Z 464.817,A -85,B 0,C 180,E1 -15590.478,E2 -15590.478} C_VEL
LIN {X 0,Y 319.806,Z 451.527,A -85,B 0,C 180,E1 -15591.132,E2 -15591.132} C_VEL
LIN {X 0,Y 320.32,Z 435.518,A -85,B 0,C 180,E1 -15591.603,E2 -15591.603} C_VEL
LIN {X 0,Y 321.673,Z 378.19,A -85,B 0,C 180,E1 -15593.022,E2 -15593.022} C_VEL
LIN {X 0,Y 316.145,Z 338.573,A -85,B 0,C 180,E1 -15594.467,E2 -15594.467} C_VEL
LIN {X 0,Y 316.749,Z 332.769,A -85,B 0,C 180,E1 -15595.989,E2 -15595.989} C_VEL
LIN {X 0,Y 315.084,Z 323.416,A -85,B 0,C 180,E1 -15598.656,E2 -15598.656} C_VEL
LIN {X 0,Y 312.513,Z 311.56,A -85,B 0,C 180,E1 -15602.239,E2 -15602.239} C_VEL
LIN {X 0,Y 312.532,Z 311.556,A -85,B 0,C 180,E1 -15605.949,E2 -15605.949} C_VEL
LIN {X 0,Y 312.504,Z 311.556,A -85,B 0,C 180,E1 -15609.027,E2 -15609.027} C_VEL
LIN {X 0,Y 312.486,Z 311.563,A -85,B 0,C 180,E1 -15612.431,E2 -15612.431} C_VEL
LIN {X 0,Y 312.454,Z 311.563,A -85,B 0,C 180,E1 -15616.034,E2 -15616.034} C_VEL
LIN {X 0,Y 312.5,Z 311.556,A -85,B 0,C 180,E1 -15619.874,E2 -15619.874} C_VEL
LIN {X 0,Y 312.534,Z 311.556,A -85,B 0,C 180,E1 -15622.616,E2 -15622.616} C_VEL
LIN {X 0,Y 312.514,Z 311.555,A -85,B 0,C 180,E1 -15626.311,E2 -15626.311} C_VEL
LIN {X 0,Y 312.533,Z 311.549,A -85,B 0,C 180,E1 -15630.349,E2 -15630.349} C_VEL
LIN {X 0,Y 312.591,Z 311.544,A -85,B 0,C 180,E1 -15634.066,E2 -15634.066} C_VEL
LIN {X 0,Y 312.582,Z 311.547,A -85,B 0,C 180,E1 -15637.529,E2 -15637.529} C_VEL
LIN {X 0,Y 312.633,Z 311.541,A -85,B 0,C 180,E1 -15641.656,E2 -15641.656} C_VEL
LIN {X 0,Y 312.688,Z 311.534,A -85,B 0,C 180,E1 -15645.686,E2 -15645.686} C_VEL
LIN {X 0,Y 312.696,Z 311.534,A -85,B 0,C 180,E1 -15649.642,E2 -15649.642} C_VEL
LIN {X 0,Y 312.866,Z 311.51,A -85,B 0,C 180,E1 -15652.254,E2 -15652.254} C_VEL
LIN {X 0,Y 312.712,Z 311.529,A -85,B 0,C 180,E1 -15654.843,E2 -15654.843} C_VEL
LIN {X 0,Y 312.985,Z 311.493,A -85,B 0,C 180,E1 -15658.714,E2 -15658.714} C_VEL
LIN {X 0,Y 312.983,Z 311.496,A -85,B 0,C 180,E1 -15661.287,E2 -15661.287} C_VEL
LIN {X 0,Y 312.703,Z 311.53,A -85,B 0,C 180,E1 -15665.158,E2 -15665.158} C_VEL
LIN {X 0,Y 312.813,Z 311.52,A -85,B 0,C 180,E1 -15667.748,E2 -15667.748} C_VEL
LIN {X 0,Y 312.664,Z 311.535,A -85,B 0,C 180,E1 -15671.672,E2 -15671.672} C_VEL
LIN {X 0,Y 312.695,Z 311.53,A -85,B 0,C 180,E1 -15674.888,E2 -15674.888} C_VEL
LIN {X 0,Y 312.605,Z 311.542,A -85,B 0,C 180,E1 -15679.226,E2 -15679.226} C_VEL
LIN {X 0,Y 312.518,Z 311.553,A -85,B 0,C 180,E1 -15682.78,E2 -15682.78} C_VEL
LIN {X 0,Y 312.527,Z 311.551,A -85,B 0,C 180,E1 -15685.909,E2 -15685.909} C_VEL
LIN {X 0,Y 312.496,Z 311.555,A -85,B 0,C 180,E1 -15689.656,E2 -15689.656} C_VEL
LIN {X 0,Y 312.516,Z 311.553,A -85,B 0,C 180,E1 -15693.69,E2 -15693.69} C_VEL
LIN {X 0,Y 312.512,Z 311.553,A -85,B 0,C 180,E1 -15697.388,E2 -15697.388} C_VEL
LIN {X 0,Y 312.486,Z 311.559,A -85,B 0,C 180,E1 -15700.71,E2 -15700.71} C_VEL
LIN {X 0,Y 312.449,Z 311.562,A -85,B 0,C 180,E1 -15704.211,E2 -15704.211} C_VEL
LIN {X 0,Y 312.453,Z 311.561,A -85,B 0,C 180,E1 -15707.926,E2 -15707.926} C_VEL
LIN {X 0,Y 312.483,Z 311.556,A -85,B 0,C 180,E1 -15711.924,E2 -15711.924} C_VEL
LIN {X 0,Y 312.53,Z 311.55,A -85,B 0,C 180,E1 -15714.221,E2 -15714.221} C_VEL
LIN {X 0,Y 312.501,Z 311.561,A -85,B 0,C 180,E1 -15717.335,E2 -15717.335} C_VEL
LIN {X 0,Y 312.505,Z 311.559,A -85,B 0,C 180,E1 -15721.293,E2 -15721.293} C_VEL
LIN {X 0,Y 312.547,Z 311.549,A -85,B 0,C 180,E1 -15724.709,E2 -15724.709} C_VEL
LIN {X 0,Y 312.564,Z 311.553,A -85,B 0,C 180,E1 -15727.528,E2 -15727.528} C_VEL
LIN {X 0,Y 312.584,Z 311.55,A -85,B 0,C 180,E1 -15731.654,E2 -15731.654} C_VEL
LIN {X 0,Y 312.689,Z 311.537,A -85,B 0,C 180,E1 -15735.687,E2 -15735.687} C_VEL
LIN {X 0,Y 312.687,Z 311.535,A -85,B 0,C 180,E1 -15739.642,E2 -15739.642} C_VEL
LIN {X 0,Y 312.799,Z 311.521,A -85,B 0,C 180,E1 -15742.253,E2 -15742.253} C_VEL
LIN {X 0,Y 312.685,Z 311.532,A -85,B 0,C 180,E1 -15744.843,E2 -15744.843} C_VEL
LIN {X 0,Y 312.966,Z 311.498,A -85,B 0,C 180,E1 -15748.714,E2 -15748.714} C_VEL
LIN {X 0,Y 312.966,Z 311.497,A -85,B 0,C 180,E1 -15751.287,E2 -15751.287} C_VEL
LIN {X 0,Y 312.844,Z 311.518,A -85,B 0,C 180,E1 -15756.45,E2 -15756.45} C_VEL
LIN {X 0,Y 312.682,Z 311.538,A -85,B 0,C 180,E1 -15760.359,E2 -15760.359} C_VEL
LIN {X 0,Y 312.608,Z 311.546,A -85,B 0,C 180,E1 -15764.821,E2 -15764.821} C_VEL
LIN {X 0,Y 312.553,Z 311.553,A -85,B 0,C 180,E1 -15769.193,E2 -15769.193} C_VEL
LIN {X 0,Y 312.57,Z 311.667,A -85,B 0,C 180,E1 -15770.913,E2 -15770.913} C_VEL
